LIN {X 0,Y 169.42,Z 430.477,A -85,B 0,C 180,E1 -24406.881,E2 -24406.881} C_VEL
LIN {X 0,Y 171.405,Z 398.166,A -85,B 0,C 180,E1 -24408.159,E2 -24408.159} C_VEL
LIN {X 0,Y 167.456,Z 387.202,A -85,B 0,C 180,E1 -24409.755,E2 -24409.755} C_VEL
LIN {X 0,Y 162.676,Z 376.705,A -85,B 0,C 180,E1 -24411.669,E2 -24411.669} C_VEL
LIN {X 0,Y 156.183,Z 365.5,A -85,B 0,C 180,E1 -24414.347,E2 -24414.347} C_VEL
LIN {X 0,Y 150.616,Z 356.98,A -85,B 0,C 180,E1 -24416.81,E2 -24416.81} C_VEL
LIN {X 0,Y 148.688,Z 354.013,A -85,B 0,C 180,E1 -24417.73,E2 -24417.73} C_VEL
LIN {X 0,Y 146.46,Z 350.663,A -85,B 0,C 180,E1 -24418.836,E2 -24418.836} C_VEL
LIN {X 0,Y 143.8,Z 347.278,A -85,B 0,C 180,E1 -24420.188,E2 -24420.188} C_VEL
LIN {X 0,Y 143.258,Z 345.674,A -85,B 0,C 180,E1 -24420.838,E2 -24420.838} C_VEL
LIN {X 0,Y 143.168,Z 345.197,A -85,B 0,C 180,E1 -24421.462,E2 -24421.462} C_VEL
LIN {X 0,Y 143.113,Z 345.14,A -85,B 0,C 180,E1 -24426.108,E2 -24426.108} C_VEL
LIN {X 0,Y 143.077,Z 345.141,A -85,B 0,C 180,E1 -24429.685,E2 -24429.685} C_VEL
LIN {X 0,Y 143.059,Z 345.139,A -85,B 0,C 180,E1 -24433.454,E2 -24433.454} C_VEL
LIN {X 0,Y 143.067,Z 345.145,A -85,B 0,C 180,E1 -24437.465,E2 -24437.465} C_VEL
LIN {X 0,Y 143.079,Z 345.123,A -85,B 0,C 180,E1 -24441.806,E2 -24441.806} C_VEL
LIN {X 0,Y 143.178,Z 345.126,A -85,B 0,C 180,E1 -24447.319,E2 -24447.319} C_VEL
LIN {X 0,Y 143.184,Z 345.102,A -85,B 0,C 180,E1 -24452.069,E2 -24452.069} C_VEL
LIN {X 0,Y 143.23,Z 345.111,A -85,B 0,C 180,E1 -24458.796,E2 -24458.796} C_VEL
LIN {X 0,Y 143.264,Z 345.082,A -85,B 0,C 180,E1 -24462.881,E2 -24462.881} C_VEL
LIN {X 0,Y 143.535,Z 345.1,A -85,B 0,C 180,E1 -24468.705,E2 -24468.705} C_VEL
LIN {X 0,Y 143.609,Z 345.048,A -85,B 0,C 180,E1 -24471.557,E2 -24471.557} C_VEL
LIN {X 0,Y 144.158,Z 345.024,A -85,B 0,C 180,E1 -24479.999,E2 -24479.999} C_VEL
LIN {X 0,Y 143.623,Z 345.077,A -85,B 0,C 180,E1 -24488.441,E2 -24488.441} C_VEL
LIN {X 0,Y 143.499,Z 345.099,A -85,B 0,C 180,E1 -24491.615,E2 -24491.615} C_VEL
LIN {X 0,Y 143.251,Z 345.109,A -85,B 0,C 180,E1 -24497.119,E2 -24497.119} C_VEL
LIN {X 0,Y 143.223,Z 345.13,A -85,B 0,C 180,E1 -24501.197,E2 -24501.197} C_VEL
LIN {X 0,Y 143.183,Z 345.151,A -85,B 0,C 180,E1 -24507.93,E2 -24507.93} C_VEL
LIN {X 0,Y 143.158,Z 345.189,A -85,B 0,C 180,E1 -24514.25,E2 -24514.25} C_VEL
LIN {X 0,Y 143.258,Z 345.961,A -85,B 0,C 180,E1 -24515.138,E2 -24515.138} C_VEL
LIN {X 0,Y 144.692,Z 348.88,A -85,B 0,C 180,E1 -24516.138,E2 -24516.138} C_VEL
LIN {X 0,Y 146.266,Z 350.451,A -85,B 0,C 180,E1 -24516.897,E2 -24516.897} C_VEL
LIN {X 0,Y 148.435,Z 353.858,A -85,B 0,C 180,E1 -24517.989,E2 -24517.989} C_VEL
LIN {X 0,Y 149.674,Z 355.677,A -85,B 0,C 180,E1 -24518.581,E2 -24518.581} C_VEL
LIN {X 0,Y 154.684,Z 363.406,A -85,B 0,C 180,E1 -24520.852,E2 -24520.852} C_VEL
LIN {X 0,Y 159.853,Z 373.317,A -85,B 0,C 180,E1 -24523.121,E2 -24523.121} C_VEL
LIN {X 0,Y 165.254,Z 385.644,A -85,B 0,C 180,E1 -24525.399,E2 -24525.399} C_VEL
LIN {X 0,Y 170.967,Z 401.167,A -85,B 0,C 180,E1 -24527.725,E2 -24527.725} C_VEL
LIN {X 0,Y 171.216,Z 402.78,A -85,B 0,C 180,E1 -24527.873,E2 -24527.873} C_VEL
LIN {X 0,Y 168.233,Z 448.35,A -85,B 0,C 180,E1 -24529.719,E2 -24529.719} C_VEL
LIN {X 0,Y 167.173,Z 458.294,A -85,B 0,C 180,E1 -24530.339,E2 -24530.339} C_VEL
LIN {X 0,Y 165.56,Z 468.543,A -85,B 0,C 180,E1 -24531.234,E2 -24531.234} C_VEL
LIN {X 0,Y 163.658,Z 477.716,A -85,B 0,C 180,E1 -24532.27,E2 -24532.27} C_VEL
LIN {X 0,Y 161.167,Z 488.501,A -85,B 0,C 180,E1 -24533.935,E2 -24533.935} C_VEL
LIN {X 0,Y 158.212,Z 498.547,A -85,B 0,C 180,E1 -24535.887,E2 -24535.887} C_VEL
LIN {X 0,Y 155.117,Z 507.96,A -85,B 0,C 180,E1 -24538.217,E2 -24538.217} C_VEL
LIN {X 0,Y 152.756,Z 515.01,A -85,B 0,C 180,E1 -24540.357,E2 -24540.357} C_VEL
LIN {X 0,Y 149.485,Z 523.905,A -85,B 0,C 180,E1 -24543.758,E2 -24543.758} C_VEL
LIN {X 0,Y 147.045,Z 530.294,A -85,B 0,C 180,E1 -24546.777,E2 -24546.777} C_VEL
LIN {X 0,Y 144.875,Z 536.086,A -85,B 0,C 180,E1 -24550.149,E2 -24550.149} C_VEL
LIN {X 0,Y 142.805,Z 541.677,A -85,B 0,C 180,E1 -24554.295,E2 -24554.295} C_VEL
LIN {X 0,Y 141.487,Z 546.063,A -85,B 0,C 180,E1 -24558.539,E2 -24558.539} C_VEL
LIN {X 0,Y 140.923,Z 548.391,A -85,B 0,C 180,E1 -24561.395,E2 -24561.395} C_VEL
LIN {X 0,Y 140.424,Z 551.696,A -85,B 0,C 180,E1 -24567.274,E2 -24567.274} C_VEL
LIN {X 0,Y 139.703,Z 552.498,A -85,B 0,C 180,E1 -24569.651,E2 -24569.651} C_VEL
LIN {X 0,Y 138.124,Z 553.012,A -85,B 0,C 180,E1 -24572.007,E2 -24572.007} C_VEL
LIN {X 0,Y 134.717,Z 553.305,A -85,B 0,C 180,E1 -24576.843,E2 -24576.843} C_VEL
LIN {X 0,Y 134.06,Z 553.015,A -85,B 0,C 180,E1 -24579.375,E2 -24579.375} C_VEL
LIN {X 0,Y 134.148,Z 552.859,A -85,B 0,C 180,E1 -24580.224,E2 -24580.224} C_VEL
LIN {X 0,Y 135.606,Z 551.577,A -85,B 0,C 180,E1 -24585.018,E2 -24585.018} C_VEL
LIN {X 0,Y 138.515,Z 548.533,A -85,B 0,C 180,E1 -24590.803,E2 -24590.803} C_VEL
LIN {X 0,Y 141.774,Z 545.076,A -85,B 0,C 180,E1 -24594.92,E2 -24594.92} C_VEL
LIN {X 0,Y 145.584,Z 540.569,A -85,B 0,C 180,E1 -24598.865,E2 -24598.865} C_VEL
LIN {X 0,Y 150.668,Z 533.867,A -85,B 0,C 180,E1 -24603.156,E2 -24603.156} C_VEL
LIN {X 0,Y 155.126,Z 527.779,A -85,B 0,C 180,E1 -24606.083,E2 -24606.083} C_VEL
LIN {X 0,Y 159.759,Z 520.62,A -85,B 0,C 180,E1 -24608.82,E2 -24608.82} C_VEL
LIN {X 0,Y 164.818,Z 511.938,A -85,B 0,C 180,E1 -24611.371,E2 -24611.371} C_VEL
LIN {X 0,Y 169.744,Z 502.444,A -85,B 0,C 180,E1 -24613.498,E2 -24613.498} C_VEL
LIN {X 0,Y 173.661,Z 493.629,A -85,B 0,C 180,E1 -24615.09,E2 -24615.09} C_VEL
LIN {X 0,Y 177.16,Z 484.552,A -85,B 0,C 180,E1 -24616.384,E2 -24616.384} C_VEL
LIN {X 0,Y 180.708,Z 473.055,A -85,B 0,C 180,E1 -24617.641,E2 -24617.641} C_VEL
LIN {X 0,Y 183.45,Z 461.877,A -85,B 0,C 180,E1 -24618.506,E2 -24618.506} C_VEL
LIN {X 0,Y 185.418,Z 450.53,A -85,B 0,C 180,E1 -24619.129,E2 -24619.129} C_VEL
LIN {X 0,Y 187.313,Z 431.246,A -85,B 0,C 180,E1 -24619.859,E2 -24619.859} C_VEL
LIN {X 0,Y 188.443,Z 418.099,A -85,B 0,C 180,E1 -24620.308,E2 -24620.308} C_VEL
LIN {X 0,Y 185.471,Z 410.111,A -85,B 0,C 180,E1 -24622.466,E2 -24622.466} C_VEL
LIN {X 0,Y 181.792,Z 401.756,A -85,B 0,C 180,E1 -24625.407,E2 -24625.407} C_VEL
LIN {X 0,Y 178.228,Z 394.65,A -85,B 0,C 180,E1 -24628.667,E2 -24628.667} C_VEL
LIN {X 0,Y 176.004,Z 390.795,A -85,B 0,C 180,E1 -24631.014,E2 -24631.014} C_VEL
LIN {X 0,Y 173.429,Z 386.846,A -85,B 0,C 180,E1 -24634.224,E2 -24634.224} C_VEL
LIN {X 0,Y 171.067,Z 383.644,A -85,B 0,C 180,E1 -24638.018,E2 -24638.018} C_VEL
LIN {X 0,Y 170.413,Z 382.188,A -85,B 0,C 180,E1 -24639.565,E2 -24639.565} C_VEL
LIN {X 0,Y 168.485,Z 380.243,A -85,B 0,C 180,E1 -24647.962,E2 -24647.962} C_VEL
LIN {X 0,Y 168.748,Z 380.458,A -85,B 0,C 180,E1 -24651.166,E2 -24651.166} C_VEL
LIN {X 0,Y 170.973,Z 382.26,A -85,B 0,C 180,E1 -24657.74,E2 -24657.74} C_VEL
LIN {X 0,Y 172.71,Z 385.701,A -85,B 0,C 180,E1 -24660.96,E2 -24660.96} C_VEL
LIN {X 0,Y 174.238,Z 387.45,A -85,B 0,C 180,E1 -24663.03,E2 -24663.03} C_VEL
LIN {X 0,Y 176.879,Z 391.787,A -85,B 0,C 180,E1 -24666.13,E2 -24666.13} C_VEL
LIN {X 0,Y 179.803,Z 396.635,A -85,B 0,C 180,E1 -24668.996,E2 -24668.996} C_VEL
LIN {X 0,Y 183.75,Z 403.362,A -85,B 0,C 180,E1 -24672.204,E2 -24672.204} C_VEL
LIN {X 0,Y 187.337,Z 411.633,A -85,B 0,C 180,E1 -24674.887,E2 -24674.887} C_VEL
LIN {X 0,Y 188.71,Z 415.167,A -85,B 0,C 180,E1 -24675.847,E2 -24675.847} C_VEL
LIN {X 0,Y 185.895,Z 445.064,A -85,B 0,C 180,E1 -24676.866,E2 -24676.866} C_VEL
LIN {X 0,Y 184.526,Z 454.52,A -85,B 0,C 180,E1 -24677.341,E2 -24677.341} C_VEL
LIN {X 0,Y 182.323,Z 464.877,A -85,B 0,C 180,E1 -24678.036,E2 -24678.036} C_VEL
LIN {X 0,Y 179.311,Z 476.023,A -85,B 0,C 180,E1 -24679.133,E2 -24679.133} C_VEL
LIN {X 0,Y 176.115,Z 485.452,A -85,B 0,C 180,E1 -24680.318,E2 -24680.318} C_VEL
LIN {X 0,Y 172.274,Z 494.993,A -85,B 0,C 180,E1 -24681.86,E2 -24681.86} C_VEL
LIN {X 0,Y 168.027,Z 504.044,A -85,B 0,C 180,E1 -24683.722,E2 -24683.722} C_VEL
LIN {X 0,Y 163.812,Z 511.888,A -85,B 0,C 180,E1 -24685.716,E2 -24685.716} C_VEL
LIN {X 0,Y 158.598,Z 520.414,A -85,B 0,C 180,E1 -24688.508,E2 -24688.508} C_VEL
LIN {X 0,Y 154.104,Z 526.971,A -85,B 0,C 180,E1 -24691.229,E2 -24691.229} C_VEL
LIN {X 0,Y 149.899,Z 532.66,A -85,B 0,C 180,E1 -24694.238,E2 -24694.238} C_VEL
LIN {X 0,Y 146.063,Z 537.442,A -85,B 0,C 180,E1 -24697.447,E2 -24697.447} C_VEL
LIN {X 0,Y 141.742,Z 542.341,A -85,B 0,C 180,E1 -24701.949,E2 -24701.949} C_VEL
LIN {X 0,Y 139.33,Z 544.911,A -85,B 0,C 180,E1 -24705.075,E2 -24705.075} C_VEL
LIN {X 0,Y 136.054,Z 547.988,A -85,B 0,C 180,E1 -24710.792,E2 -24710.792} C_VEL
LIN {X 0,Y 134.497,Z 549.246,A -85,B 0,C 180,E1 -24714.915,E2 -24714.915} C_VEL
LIN {X 0,Y 133.629,Z 549.592,A -85,B 0,C 180,E1 -24718.269,E2 -24718.269} C_VEL
LIN {X 0,Y 132.836,Z 549.037,A -85,B 0,C 180,E1 -24724.96,E2 -24724.96} C_VEL
LIN {X 0,Y 132.855,Z 547.969,A -85,B 0,C 180,E1 -24728.266,E2 -24728.266} C_VEL
LIN {X 0,Y 133.226,Z 546.339,A -85,B 0,C 180,E1 -24731.723,E2 -24731.723} C_VEL
LIN {X 0,Y 134.201,Z 543.282,A -85,B 0,C 180,E1 -24736.37,E2 -24736.37} C_VEL
LIN {X 0,Y 135.436,Z 539.701,A -85,B 0,C 180,E1 -24740.384,E2 -24740.384} C_VEL
LIN {X 0,Y 137.031,Z 535.472,A -85,B 0,C 180,E1 -24744.113,E2 -24744.113} C_VEL
LIN {X 0,Y 139.182,Z 530.061,A -85,B 0,C 180,E1 -24747.902,E2 -24747.902} C_VEL
LIN {X 0,Y 141.754,Z 523.767,A -85,B 0,C 180,E1 -24751.421,E2 -24751.421} C_VEL
LIN {X 0,Y 144.817,Z 515.992,A -85,B 0,C 180,E1 -24754.872,E2 -24754.872} C_VEL
LIN {X 0,Y 147.942,Z 507.566,A -85,B 0,C 180,E1 -24757.85,E2 -24757.85} C_VEL
LIN {X 0,Y 150.993,Z 499.018,A -85,B 0,C 180,E1 -24760.252,E2 -24760.252} C_VEL
LIN {X 0,Y 153.669,Z 490.48,A -85,B 0,C 180,E1 -24762.212,E2 -24762.212} C_VEL
LIN {X 0,Y 156.274,Z 480.837,A -85,B 0,C 180,E1 -24763.989,E2 -24763.989} C_VEL
LIN {X 0,Y 158.85,Z 469.502,A -85,B 0,C 180,E1 -24765.575,E2 -24765.575} C_VEL
LIN {X 0,Y 160.694,Z 458.708,A -85,B 0,C 180,E1 -24766.72,E2 -24766.72} C_VEL
LIN {X 0,Y 162.232,Z 447.473,A -85,B 0,C 180,E1 -24767.521,E2 -24767.521} C_VEL
LIN {X 0,Y 163.725,Z 428.996,A -85,B 0,C 180,E1 -24768.341,E2 -24768.341} C_VEL
LIN {X 0,Y 165.514,Z 399.768,A -85,B 0,C 180,E1 -24769.546,E2 -24769.546} C_VEL
LIN {X 0,Y 161.92,Z 389.844,A -85,B 0,C 180,E1 -24771.101,E2 -24771.101} C_VEL
LIN {X 0,Y 157.712,Z 380.464,A -85,B 0,C 180,E1 -24772.916,E2 -24772.916} C_VEL
LIN {X 0,Y 151.583,Z 369.812,A -85,B 0,C 180,E1 -24775.593,E2 -24775.593} C_VEL
LIN {X 0,Y 145.009,Z 359.507,A -85,B 0,C 180,E1 -24778.765,E2 -24778.765} C_VEL
LIN {X 0,Y 141.709,Z 354.853,A -85,B 0,C 180,E1 -24780.492,E2 -24780.492} C_VEL
LIN {X 0,Y 139.638,Z 351.74,A -85,B 0,C 180,E1 -24781.645,E2 -24781.645} C_VEL
LIN {X 0,Y 138.864,Z 350.808,A -85,B 0,C 180,E1 -24782.071,E2 -24782.071} C_VEL
LIN {X 0,Y 136.849,Z 348.327,A -85,B 0,C 180,E1 -24783.225,E2 -24783.225} C_VEL
LIN {X 0,Y 136.198,Z 346.577,A -85,B 0,C 180,E1 -24783.99,E2 -24783.99} C_VEL
LIN {X 0,Y 136.082,Z 346.085,A -85,B 0,C 180,E1 -24784.618,E2 -24784.618} C_VEL
LIN {X 0,Y 136.053,Z 346.02,A -85,B 0,C 180,E1 -24789.208,E2 -24789.208} C_VEL
LIN {X 0,Y 136.001,Z 346.019,A -85,B 0,C 180,E1 -24793.658,E2 -24793.658} C_VEL
LIN {X 0,Y 136.007,Z 346.018,A -85,B 0,C 180,E1 -24797.796,E2 -24797.796} C_VEL
LIN {X 0,Y 136.028,Z 346,A -85,B 0,C 180,E1 -24801.684,E2 -24801.684} C_VEL
LIN {X 0,Y 136.085,Z 346.032,A -85,B 0,C 180,E1 -24805.722,E2 -24805.722} C_VEL
LIN {X 0,Y 136.125,Z 345.982,A -85,B 0,C 180,E1 -24812.311,E2 -24812.311} C_VEL
LIN {X 0,Y 136.196,Z 345.984,A -85,B 0,C 180,E1 -24818.824,E2 -24818.824} C_VEL
LIN {X 0,Y 136.234,Z 345.98,A -85,B 0,C 180,E1 -24825.051,E2 -24825.051} C_VEL
LIN {X 0,Y 136.427,Z 345.989,A -85,B 0,C 180,E1 -24828.177,E2 -24828.177} C_VEL
LIN {X 0,Y 136.538,Z 345.933,A -85,B 0,C 180,E1 -24831.116,E2 -24831.116} C_VEL
LIN {X 0,Y 137.115,Z 345.901,A -85,B 0,C 180,E1 -24839.999,E2 -24839.999} C_VEL
LIN {X 0,Y 136.549,Z 345.964,A -85,B 0,C 180,E1 -24848.882,E2 -24848.882} C_VEL
LIN {X 0,Y 136.414,Z 345.975,A -85,B 0,C 180,E1 -24851.892,E2 -24851.892} C_VEL
LIN {X 0,Y 136.165,Z 346.002,A -85,B 0,C 180,E1 -24858.039,E2 -24858.039} C_VEL
LIN {X 0,Y 136.148,Z 346.003,A -85,B 0,C 180,E1 -24861.694,E2 -24861.694} C_VEL
LIN {X 0,Y 136.092,Z 346.024,A -85,B 0,C 180,E1 -24868.608,E2 -24868.608} C_VEL
LIN {X 0,Y 136.09,Z 346.281,A -85,B 0,C 180,E1 -24871.525,E2 -24871.525} C_VEL
LIN {X 0,Y 136.445,Z 347.466,A -85,B 0,C 180,E1 -24872.302,E2 -24872.302} C_VEL
LIN {X 0,Y 138.171,Z 350.216,A -85,B 0,C 180,E1 -24873.384,E2 -24873.384} C_VEL
LIN {X 0,Y 139.409,Z 351.47,A -85,B 0,C 180,E1 -24874.054,E2 -24874.054} C_VEL
LIN {X 0,Y 141.532,Z 354.861,A -85,B 0,C 180,E1 -24875.257,E2 -24875.257} C_VEL
LIN {X 0,Y 143.129,Z 357.003,A -85,B 0,C 180,E1 -24876.101,E2 -24876.101} C_VEL
LIN {X 0,Y 148.206,Z 364.638,A -85,B 0,C 180,E1 -24878.667,E2 -24878.667} C_VEL
LIN {X 0,Y 152.246,Z 371.513,A -85,B 0,C 180,E1 -24880.573,E2 -24880.573} C_VEL
LIN {X 0,Y 157.962,Z 383.796,A -85,B 0,C 180,E1 -24883.197,E2 -24883.197} C_VEL
LIN {X 0,Y 163.187,Z 397.335,A -85,B 0,C 180,E1 -24885.518,E2 -24885.518} C_VEL
LIN {X 0,Y 165.396,Z 403.646,A -85,B 0,C 180,E1 -24886.469,E2 -24886.469} C_VEL
LIN {X 0,Y 162.325,Z 448.845,A -85,B 0,C 180,E1 -24888.358,E2 -24888.358} C_VEL
LIN {X 0,Y 161.232,Z 458.516,A -85,B 0,C 180,E1 -24888.987,E2 -24888.987} C_VEL
LIN {X 0,Y 159.578,Z 468.651,A -85,B 0,C 180,E1 -24889.901,E2 -24889.901} C_VEL
LIN {X 0,Y 157.602,Z 477.772,A -85,B 0,C 180,E1 -24890.958,E2 -24890.958} C_VEL
LIN {X 0,Y 155.005,Z 488.528,A -85,B 0,C 180,E1 -24892.668,E2 -24892.668} C_VEL
LIN {X 0,Y 151.935,Z 498.551,A -85,B 0,C 180,E1 -24894.675,E2 -24894.675} C_VEL
LIN {X 0,Y 148.705,Z 507.945,A -85,B 0,C 180,E1 -24897.077,E2 -24897.077} C_VEL
LIN {X 0,Y 145.899,Z 515.846,A -85,B 0,C 180,E1 -24899.616,E2 -24899.616} C_VEL
LIN {X 0,Y 142.775,Z 523.96,A -85,B 0,C 180,E1 -24902.871,E2 -24902.871} C_VEL
LIN {X 0,Y 139.995,Z 530.839,A -85,B 0,C 180,E1 -24906.321,E2 -24906.321} C_VEL
LIN {X 0,Y 138.164,Z 535.532,A -85,B 0,C 180,E1 -24909.141,E2 -24909.141} C_VEL
LIN {X 0,Y 135.935,Z 541.224,A -85,B 0,C 180,E1 -24913.479,E2 -24913.479} C_VEL
LIN {X 0,Y 134.51,Z 545.696,A -85,B 0,C 180,E1 -24917.936,E2 -24917.936} C_VEL
LIN {X 0,Y 133.889,Z 548.023,A -85,B 0,C 180,E1 -24920.939,E2 -24920.939} C_VEL
LIN {X 0,Y 133.332,Z 551.432,A -85,B 0,C 180,E1 -24926.978,E2 -24926.978} C_VEL
LIN {X 0,Y 133.415,Z 552.393,A -85,B 0,C 180,E1 -24930,E2 -24930} C_VEL
LIN {X 0,Y 133.515,Z 553.311,A -85,B 0,C 180,E1 -24936.043,E2 -24936.043} C_VEL
LIN {X 0,Y 134.148,Z 552.859,A -85,B 0,C 180,E1 -24940.224,E2 -24940.224} C_VEL
LIN {X 0,Y 134.121,Z 552.393,A -85,B 0,C 180,E1 -24942.742,E2 -24942.742} C_VEL
LIN {X 0,Y 132.78,Z 551.096,A -85,B 0,C 180,E1 -24946.934,E2 -24946.934} C_VEL
LIN {X 0,Y 132.116,Z 549.103,A -85,B 0,C 180,E1 -24951.129,E2 -24951.129} C_VEL
LIN {X 0,Y 133.122,Z 547.442,A -85,B 0,C 180,E1 -24953.54,E2 -24953.54} C_VEL
LIN {X 0,Y 136.723,Z 543.887,A -85,B 0,C 180,E1 -24957.557,E2 -24957.557} C_VEL
LIN {X 0,Y 140.881,Z 539.102,A -85,B 0,C 180,E1 -24961.587,E2 -24961.587} C_VEL
LIN {X 0,Y 145.729,Z 533.082,A -85,B 0,C 180,E1 -24965.36,E2 -24965.36} C_VEL
LIN {X 0,Y 150.396,Z 527.009,A -85,B 0,C 180,E1 -24968.255,E2 -24968.255} C_VEL
LIN {X 0,Y 155.42,Z 519.728,A -85,B 0,C 180,E1 -24970.971,E2 -24970.971} C_VEL
LIN {X 0,Y 160.705,Z 510.929,A -85,B 0,C 180,E1 -24973.534,E2 -24973.534} C_VEL
LIN {X 0,Y 165.299,Z 502.475,A -85,B 0,C 180,E1 -24975.41,E2 -24975.41} C_VEL
LIN {X 0,Y 169.386,Z 493.684,A -85,B 0,C 180,E1 -24976.994,E2 -24976.994} C_VEL
LIN {X 0,Y 173.603,Z 482.834,A -85,B 0,C 180,E1 -24978.498,E2 -24978.498} C_VEL
LIN {X 0,Y 176.583,Z 473.688,A -85,B 0,C 180,E1 -24979.474,E2 -24979.474} C_VEL
LIN {X 0,Y 179.612,Z 461.78,A -85,B 0,C 180,E1 -24980.392,E2 -24980.392} C_VEL
LIN {X 0,Y 181.585,Z 450.908,A -85,B 0,C 180,E1 -24980.988,E2 -24980.988} C_VEL
LIN {X 0,Y 183.476,Z 432.692,A -85,B 0,C 180,E1 -24981.682,E2 -24981.682} C_VEL
LIN {X 0,Y 184.515,Z 420.712,A -85,B 0,C 180,E1 -24982.108,E2 -24982.108} C_VEL
LIN {X 0,Y 181.36,Z 412.254,A -85,B 0,C 180,E1 -24984.694,E2 -24984.694} C_VEL
LIN {X 0,Y 178.028,Z 404.613,A -85,B 0,C 180,E1 -24987.713,E2 -24987.713} C_VEL
LIN {X 0,Y 175.056,Z 398.582,A -85,B 0,C 180,E1 -24990.874,E2 -24990.874} C_VEL
LIN {X 0,Y 173.509,Z 396.227,A -85,B 0,C 180,E1 -24992.688,E2 -24992.688} C_VEL
LIN {X 0,Y 171.894,Z 393.442,A -85,B 0,C 180,E1 -24994.974,E2 -24994.974} C_VEL
LIN {X 0,Y 169.789,Z 390.364,A -85,B 0,C 180,E1 -24998.654,E2 -24998.654} C_VEL
LIN {X 0,Y 169.326,Z 389.162,A -85,B 0,C 180,E1 -24999.853,E2 -24999.853} C_VEL
LIN {X 0,Y 167.545,Z 387.302,A -85,B 0,C 180,E1 -25007.894,E2 -25007.894} C_VEL
LIN {X 0,Y 167.798,Z 387.503,A -85,B 0,C 180,E1 -25011.116,E2 -25011.116} C_VEL
LIN {X 0,Y 169.735,Z 389.122,A -85,B 0,C 180,E1 -25017.182,E2 -25017.182} C_VEL
LIN {X 0,Y 171.478,Z 392.631,A -85,B 0,C 180,E1 -25020.605,E2 -25020.605} C_VEL
LIN {X 0,Y 172.688,Z 394.127,A -85,B 0,C 180,E1 -25022.333,E2 -25022.333} C_VEL
LIN {X 0,Y 175.084,Z 398.253,A -85,B 0,C 180,E1 -25025.358,E2 -25025.358} C_VEL
LIN {X 0,Y 177.855,Z 403.08,A -85,B 0,C 180,E1 -25028.234,E2 -25028.234} C_VEL
LIN {X 0,Y 181.051,Z 408.824,A -85,B 0,C 180,E1 -25031.037,E2 -25031.037} C_VEL
LIN {X 0,Y 184.2,Z 416.496,A -85,B 0,C 180,E1 -25033.615,E2 -25033.615} C_VEL
LIN {X 0,Y 184.757,Z 418.082,A -85,B 0,C 180,E1 -25034.057,E2 -25034.057} C_VEL
LIN {X 0,Y 182.12,Z 445.2,A -85,B 0,C 180,E1 -25034.994,E2 -25034.994} C_VEL
LIN {X 0,Y 180.59,Z 455.19,A -85,B 0,C 180,E1 -25035.496,E2 -25035.496} C_VEL
LIN {X 0,Y 178.403,Z 465.096,A -85,B 0,C 180,E1 -25036.162,E2 -25036.162} C_VEL
LIN {X 0,Y 175.245,Z 476.308,A -85,B 0,C 180,E1 -25037.26,E2 -25037.26} C_VEL
LIN {X 0,Y 172.143,Z 485.121,A -85,B 0,C 180,E1 -25038.338,E2 -25038.338} C_VEL
LIN {X 0,Y 167.782,Z 495.487,A -85,B 0,C 180,E1 -25040.013,E2 -25040.013} C_VEL
LIN {X 0,Y 163.619,Z 503.956,A -85,B 0,C 180,E1 -25041.741,E2 -25041.741} C_VEL
LIN {X 0,Y 159.181,Z 511.899,A -85,B 0,C 180,E1 -25043.774,E2 -25043.774} C_VEL
LIN {X 0,Y 153.572,Z 520.561,A -85,B 0,C 180,E1 -25046.628,E2 -25046.628} C_VEL
LIN {X 0,Y 149.027,Z 526.848,A -85,B 0,C 180,E1 -25049.256,E2 -25049.256} C_VEL
LIN {X 0,Y 144.444,Z 532.653,A -85,B 0,C 180,E1 -25052.359,E2 -25052.359} C_VEL
LIN {X 0,Y 139.573,Z 538.241,A -85,B 0,C 180,E1 -25056.327,E2 -25056.327} C_VEL
LIN {X 0,Y 136.454,Z 541.627,A -85,B 0,C 180,E1 -25059.415,E2 -25059.415} C_VEL
LIN {X 0,Y 133.247,Z 544.766,A -85,B 0,C 180,E1 -25063.29,E2 -25063.29} C_VEL
LIN {X 0,Y 129.46,Z 548.058,A -85,B 0,C 180,E1 -25069.467,E2 -25069.467} C_VEL
LIN {X 0,Y 128.013,Z 549.08,A -85,B 0,C 180,E1 -25072.85,E2 -25072.85} C_VEL
LIN {X 0,Y 126.957,Z 549.594,A -85,B 0,C 180,E1 -25076.388,E2 -25076.388} C_VEL
LIN {X 0,Y 126.176,Z 549.719,A -85,B 0,C 180,E1 -25079.914,E2 -25079.914} C_VEL
LIN {X 0,Y 125.801,Z 549.344,A -85,B 0,C 180,E1 -25083.454,E2 -25083.454} C_VEL
LIN {X 0,Y 125.943,Z 547.072,A -85,B 0,C 180,E1 -25090.439,E2 -25090.439} C_VEL
LIN {X 0,Y 126.87,Z 544.129,A -85,B 0,C 180,E1 -25095.566,E2 -25095.566} C_VEL
LIN {X 0,Y 127.789,Z 541.636,A -85,B 0,C 180,E1 -25098.904,E2 -25098.904} C_VEL
LIN {X 0,Y 129.998,Z 535.778,A -85,B 0,C 180,E1 -25104.571,E2 -25104.571} C_VEL
LIN {X 0,Y 132.201,Z 530.534,A -85,B 0,C 180,E1 -25108.477,E2 -25108.477} C_VEL
LIN {X 0,Y 134.983,Z 524.035,A -85,B 0,C 180,E1 -25112.305,E2 -25112.305} C_VEL
LIN {X 0,Y 138.151,Z 516.445,A -85,B 0,C 180,E1 -25115.84,E2 -25115.84} C_VEL
LIN {X 0,Y 141.565,Z 507.662,A -85,B 0,C 180,E1 -25119.069,E2 -25119.069} C_VEL
LIN {X 0,Y 144.745,Z 499.104,A -85,B 0,C 180,E1 -25121.554,E2 -25121.554} C_VEL
LIN {X 0,Y 147.786,Z 489.659,A -85,B 0,C 180,E1 -25123.756,E2 -25123.756} C_VEL
LIN {X 0,Y 150.559,Z 479.769,A -85,B 0,C 180,E1 -25125.57,E2 -25125.57} C_VEL
LIN {X 0,Y 152.965,Z 469.48,A -85,B 0,C 180,E1 -25127.032,E2 -25127.032} C_VEL
LIN {X 0,Y 154.859,Z 458.89,A -85,B 0,C 180,E1 -25128.181,E2 -25128.181} C_VEL
LIN {X 0,Y 156.412,Z 448.069,A -85,B 0,C 180,E1 -25128.978,E2 -25128.978} C_VEL
LIN {X 0,Y 157.946,Z 430.09,A -85,B 0,C 180,E1 -25129.8,E2 -25129.8} C_VEL
LIN {X 0,Y 159.769,Z 401.488,A -85,B 0,C 180,E1 -25131.012,E2 -25131.012} C_VEL
LIN {X 0,Y 155.979,Z 391.113,A -85,B 0,C 180,E1 -25132.78,E2 -25132.78} C_VEL
LIN {X 0,Y 152.062,Z 382.89,A -85,B 0,C 180,E1 -25134.555,E2 -25134.555} C_VEL
LIN {X 0,Y 146.807,Z 373.79,A -85,B 0,C 180,E1 -25137.033,E2 -25137.033} C_VEL
LIN {X 0,Y 141.181,Z 364.71,A -85,B 0,C 180,E1 -25139.948,E2 -25139.948} C_VEL
LIN {X 0,Y 137.751,Z 359.893,A -85,B 0,C 180,E1 -25141.842,E2 -25141.842} C_VEL
LIN {X 0,Y 135.354,Z 356.36,A -85,B 0,C 180,E1 -25143.273,E2 -25143.273} C_VEL
LIN {X 0,Y 133.051,Z 353.187,A -85,B 0,C 180,E1 -25144.718,E2 -25144.718} C_VEL
LIN {X 0,Y 132.328,Z 352.128,A -85,B 0,C 180,E1 -25145.197,E2 -25145.197} C_VEL
LIN {X 0,Y 130.053,Z 349.935,A -85,B 0,C 180,E1 -25146.666,E2 -25146.666} C_VEL
LIN {X 0,Y 129.128,Z 347.688,A -85,B 0,C 180,E1 -25147.641,E2 -25147.641} C_VEL
LIN {X 0,Y 129.016,Z 346.961,A -85,B 0,C 180,E1 -25148.541,E2 -25148.541} C_VEL
LIN {X 0,Y 128.924,Z 346.919,A -85,B 0,C 180,E1 -25155.127,E2 -25155.127} C_VEL
LIN {X 0,Y 128.944,Z 346.879,A -85,B 0,C 180,E1 -25159.735,E2 -25159.735} C_VEL
LIN {X 0,Y 128.982,Z 346.916,A -85,B 0,C 180,E1 -25164.818,E2 -25164.818} C_VEL
LIN {X 0,Y 129.018,Z 346.859,A -85,B 0,C 180,E1 -25170.642,E2 -25170.642} C_VEL
LIN {X 0,Y 129.016,Z 346.89,A -85,B 0,C 180,E1 -25174.164,E2 -25174.164} C_VEL
LIN {X 0,Y 129.075,Z 346.888,A -85,B 0,C 180,E1 -25177.765,E2 -25177.765} C_VEL
LIN {X 0,Y 129.154,Z 346.849,A -85,B 0,C 180,E1 -25184.211,E2 -25184.211} C_VEL
LIN {X 0,Y 129.347,Z 346.871,A -85,B 0,C 180,E1 -25187.967,E2 -25187.967} C_VEL
LIN {X 0,Y 129.464,Z 346.819,A -85,B 0,C 180,E1 -25190.627,E2 -25190.627} C_VEL
LIN {X 0,Y 130.07,Z 346.778,A -85,B 0,C 180,E1 -25199.999,E2 -25199.999} C_VEL
LIN {X 0,Y 129.471,Z 346.852,A -85,B 0,C 180,E1 -25209.371,E2 -25209.371} C_VEL
LIN {X 0,Y 129.298,Z 346.85,A -85,B 0,C 180,E1 -25212.557,E2 -25212.557} C_VEL
LIN {X 0,Y 129.084,Z 346.9,A -85,B 0,C 180,E1 -25219.066,E2 -25219.066} C_VEL
LIN {X 0,Y 129.045,Z 346.88,A -85,B 0,C 180,E1 -25222.409,E2 -25222.409} C_VEL
LIN {X 0,Y 129.095,Z 347.029,A -85,B 0,C 180,E1 -25227.563,E2 -25227.563} C_VEL
LIN {X 0,Y 129.358,Z 348.214,A -85,B 0,C 180,E1 -25228.533,E2 -25228.533} C_VEL
LIN {X 0,Y 130.768,Z 350.777,A -85,B 0,C 180,E1 -25229.647,E2 -25229.647} C_VEL
LIN {X 0,Y 132.707,Z 352.512,A -85,B 0,C 180,E1 -25230.866,E2 -25230.866} C_VEL
LIN {X 0,Y 134.929,Z 355.991,A -85,B 0,C 180,E1 -25232.311,E2 -25232.311} C_VEL
LIN {X 0,Y 136.097,Z 357.553,A -85,B 0,C 180,E1 -25233.013,E2 -25233.013} C_VEL
LIN {X 0,Y 141.892,Z 366.04,A -85,B 0,C 180,E1 -25236.274,E2 -25236.274} C_VEL
LIN {X 0,Y 147.239,Z 374.845,A -85,B 0,C 180,E1 -25239.029,E2 -25239.029} C_VEL
LIN {X 0,Y 153.048,Z 387.457,A -85,B 0,C 180,E1 -25241.892,E2 -25241.892} C_VEL
LIN {X 0,Y 158.407,Z 401.74,A -85,B 0,C 180,E1 -25244.437,E2 -25244.437} C_VEL
LIN {X 0,Y 159.627,Z 405.36,A -85,B 0,C 180,E1 -25245.007,E2 -25245.007} C_VEL
LIN {X 0,Y 158.009,Z 430.26,A -85,B 0,C 180,E1 -25246.053,E2 -25246.053} C_VEL
LIN {X 0,Y 156.427,Z 450.314,A -85,B 0,C 180,E1 -25246.959,E2 -25246.959} C_VEL
LIN {X 0,Y 155.189,Z 460.064,A -85,B 0,C 180,E1 -25247.651,E2 -25247.651} C_VEL
LIN {X 0,Y 153.42,Z 469.897,A -85,B 0,C 180,E1 -25248.595,E2 -25248.595} C_VEL
LIN {X 0,Y 151.111,Z 479.645,A -85,B 0,C 180,E1 -25249.81,E2 -25249.81} C_VEL
LIN {X 0,Y 148.921,Z 488.522,A -85,B 0,C 180,E1 -25251.295,E2 -25251.295} C_VEL
LIN {X 0,Y 146.16,Z 497.288,A -85,B 0,C 180,E1 -25253.054,E2 -25253.054} C_VEL
LIN {X 0,Y 142.801,Z 506.887,A -85,B 0,C 180,E1 -25255.529,E2 -25255.529} C_VEL
LIN {X 0,Y 139.77,Z 514.938,A -85,B 0,C 180,E1 -25258.131,E2 -25258.131} C_VEL
LIN {X 0,Y 136.237,Z 523.593,A -85,B 0,C 180,E1 -25261.692,E2 -25261.692} C_VEL
LIN {X 0,Y 133.479,Z 530.184,A -85,B 0,C 180,E1 -25265.088,E2 -25265.088} C_VEL
LIN {X 0,Y 131.517,Z 534.929,A -85,B 0,C 180,E1 -25268.033,E2 -25268.033} C_VEL
LIN {X 0,Y 129.105,Z 540.75,A -85,B 0,C 180,E1 -25272.578,E2 -25272.578} C_VEL
LIN {X 0,Y 127.558,Z 545.318,A -85,B 0,C 180,E1 -25277.268,E2 -25277.268} C_VEL
LIN {X 0,Y 126.877,Z 547.653,A -85,B 0,C 180,E1 -25280.434,E2 -25280.434} C_VEL
LIN {X 0,Y 126.246,Z 551.192,A -85,B 0,C 180,E1 -25286.808,E2 -25286.808} C_VEL
LIN {X 0,Y 126.317,Z 552.181,A -85,B 0,C 180,E1 -25290,E2 -25290} C_VEL
LIN {X 0,Y 126.301,Z 552.877,A -85,B 0,C 180,E1 -25293.19,E2 -25293.19} C_VEL
LIN {X 0,Y 126.45,Z 553.175,A -85,B 0,C 180,E1 -25296.382,E2 -25296.382} C_VEL
LIN {X 0,Y 127.659,Z 552.569,A -85,B 0,C 180,E1 -25302.721,E2 -25302.721} C_VEL
LIN {X 0,Y 130.135,Z 550.298,A -85,B 0,C 180,E1 -25308.907,E2 -25308.907} C_VEL
LIN {X 0,Y 132.977,Z 547.592,A -85,B 0,C 180,E1 -25313.352,E2 -25313.352} C_VEL
LIN {X 0,Y 133.122,Z 547.442,A -85,B 0,C 180,E1 -25313.54,E2 -25313.54} C_VEL
LIN {X 0,Y 134.341,Z 545.697,A -85,B 0,C 180,E1 -25315.886,E2 -25315.886} C_VEL
LIN {X 0,Y 135.038,Z 542.326,A -85,B 0,C 180,E1 -25319.858,E2 -25319.858} C_VEL
LIN {X 0,Y 135.842,Z 539.39,A -85,B 0,C 180,E1 -25322.957,E2 -25322.957} C_VEL
LIN {X 0,Y 137.381,Z 536.737,A -85,B 0,C 180,E1 -25325.094,E2 -25325.094} C_VEL
LIN {X 0,Y 138.168,Z 535.792,A -85,B 0,C 180,E1 -25325.742,E2 -25325.742} C_VEL
LIN {X 0,Y 144.924,Z 527.69,A -85,B 0,C 180,E1 -25329.982,E2 -25329.982} C_VEL
LIN {X 0,Y 150.177,Z 520.561,A -85,B 0,C 180,E1 -25332.732,E2 -25332.732} C_VEL
LIN {X 0,Y 155.68,Z 511.945,A -85,B 0,C 180,E1 -25335.317,E2 -25335.317} C_VEL
LIN {X 0,Y 161.051,Z 502.506,A -85,B 0,C 180,E1 -25337.425,E2 -25337.425} C_VEL
LIN {X 0,Y 165.308,Z 493.74,A -85,B 0,C 180,E1 -25338.993,E2 -25338.993} C_VEL
LIN {X 0,Y 169.688,Z 482.96,A -85,B 0,C 180,E1 -25340.479,E2 -25340.479} C_VEL
LIN {X 0,Y 173.029,Z 473.013,A -85,B 0,C 180,E1 -25341.514,E2 -25341.514} C_VEL
LIN {X 0,Y 176.051,Z 461.469,A -85,B 0,C 180,E1 -25342.38,E2 -25342.38} C_VEL
LIN {X 0,Y 178.062,Z 450.767,A -85,B 0,C 180,E1 -25342.955,E2 -25342.955} C_VEL
LIN {X 0,Y 180.02,Z 432.886,A -85,B 0,C 180,E1 -25343.626,E2 -25343.626} C_VEL
LIN {X 0,Y 180.813,Z 423.539,A -85,B 0,C 180,E1 -25343.994,E2 -25343.994} C_VEL
LIN {X 0,Y 178.175,Z 416.369,A -85,B 0,C 180,E1 -25346.38,E2 -25346.38} C_VEL
LIN {X 0,Y 175.543,Z 409.985,A -85,B 0,C 180,E1 -25349.06,E2 -25349.06} C_VEL
LIN {X 0,Y 173.161,Z 404.746,A -85,B 0,C 180,E1 -25351.833,E2 -25351.833} C_VEL
LIN {X 0,Y 170.439,Z 400.163,A -85,B 0,C 180,E1 -25355.648,E2 -25355.648} C_VEL
LIN {X 0,Y 168.378,Z 396.657,A -85,B 0,C 180,E1 -25359.721,E2 -25359.721} C_VEL
LIN {X 0,Y 168.109,Z 396.046,A -85,B 0,C 180,E1 -25360.462,E2 -25360.462} C_VEL
LIN {X 0,Y 166.609,Z 394.333,A -85,B 0,C 180,E1 -25367.825,E2 -25367.825} C_VEL
LIN {X 0,Y 166.85,Z 394.532,A -85,B 0,C 180,E1 -25371.065,E2 -25371.065} C_VEL
LIN {X 0,Y 168.548,Z 396.094,A -85,B 0,C 180,E1 -25376.714,E2 -25376.714} C_VEL
LIN {X 0,Y 170.322,Z 399.643,A -85,B 0,C 180,E1 -25380.352,E2 -25380.352} C_VEL
LIN {X 0,Y 171.28,Z 400.987,A -85,B 0,C 180,E1 -25381.796,E2 -25381.796} C_VEL
LIN {X 0,Y 173.454,Z 404.973,A -85,B 0,C 180,E1 -25384.731,E2 -25384.731} C_VEL
LIN {X 0,Y 176.085,Z 409.753,A -85,B 0,C 180,E1 -25387.599,E2 -25387.599} C_VEL
LIN {X 0,Y 178.682,Z 414.897,A -85,B 0,C 180,E1 -25390.07,E2 -25390.07} C_VEL
LIN {X 0,Y 181.098,Z 421.021,A -85,B 0,C 180,E1 -25392.199,E2 -25392.199} C_VEL
LIN {X 0,Y 178.518,Z 446.025,A -85,B 0,C 180,E1 -25393.066,E2 -25393.066} C_VEL
LIN {X 0,Y 177.024,Z 455.271,A -85,B 0,C 180,E1 -25393.528,E2 -25393.528} C_VEL
LIN {X 0,Y 175.003,Z 464.336,A -85,B 0,C 180,E1 -25394.117,E2 -25394.117} C_VEL
LIN {X 0,Y 171.612,Z 475.961,A -85,B 0,C 180,E1 -25395.214,E2 -25395.214} C_VEL
LIN {X 0,Y 168.398,Z 484.846,A -85,B 0,C 180,E1 -25396.283,E2 -25396.283} C_VEL
LIN {X 0,Y 163.708,Z 495.516,A -85,B 0,C 180,E1 -25397.98,E2 -25397.98} C_VEL
LIN {X 0,Y 158.836,Z 504.894,A -85,B 0,C 180,E1 -25399.907,E2 -25399.907} C_VEL
LIN {X 0,Y 154.585,Z 512.129,A -85,B 0,C 180,E1 -25401.77,E2 -25401.77} C_VEL
LIN {X 0,Y 148.791,Z 520.665,A -85,B 0,C 180,E1 -25404.598,E2 -25404.598} C_VEL
LIN {X 0,Y 144.148,Z 526.773,A -85,B 0,C 180,E1 -25407.154,E2 -25407.154} C_VEL
LIN {X 0,Y 138.816,Z 533.08,A -85,B 0,C 180,E1 -25410.608,E2 -25410.608} C_VEL
LIN {X 0,Y 133.569,Z 538.658,A -85,B 0,C 180,E1 -25414.741,E2 -25414.741} C_VEL
LIN {X 0,Y 129.882,Z 542.313,A -85,B 0,C 180,E1 -25418.316,E2 -25418.316} C_VEL
LIN {X 0,Y 125.738,Z 545.941,A -85,B 0,C 180,E1 -25423.397,E2 -25423.397} C_VEL
LIN {X 0,Y 122.926,Z 548.133,A -85,B 0,C 180,E1 -25428.009,E2 -25428.009} C_VEL
LIN {X 0,Y 120.191,Z 549.658,A -85,B 0,C 180,E1 -25434.949,E2 -25434.949} C_VEL
LIN {X 0,Y 119.404,Z 549.905,A -85,B 0,C 180,E1 -25438.013,E2 -25438.013} C_VEL
LIN {X 0,Y 118.742,Z 549.473,A -85,B 0,C 180,E1 -25442.601,E2 -25442.601} C_VEL
LIN {X 0,Y 118.715,Z 547.688,A -85,B 0,C 180,E1 -25449.194,E2 -25449.194} C_VEL
LIN {X 0,Y 119.525,Z 544.964,A -85,B 0,C 180,E1 -25454.657,E2 -25454.657} C_VEL
LIN {X 0,Y 121.134,Z 540.603,A -85,B 0,C 180,E1 -25460.514,E2 -25460.514} C_VEL
LIN {X 0,Y 123.002,Z 536.061,A -85,B 0,C 180,E1 -25465.084,E2 -25465.084} C_VEL
LIN {X 0,Y 125.295,Z 530.861,A -85,B 0,C 180,E1 -25469.197,E2 -25469.197} C_VEL
LIN {X 0,Y 128.134,Z 524.548,A -85,B 0,C 180,E1 -25473.145,E2 -25473.145} C_VEL
LIN {X 0,Y 131.519,Z 516.876,A -85,B 0,C 180,E1 -25476.906,E2 -25476.906} C_VEL
LIN {X 0,Y 135.039,Z 508.281,A -85,B 0,C 180,E1 -25480.225,E2 -25480.225} C_VEL
LIN {X 0,Y 138.391,Z 499.688,A -85,B 0,C 180,E1 -25482.837,E2 -25482.837} C_VEL
LIN {X 0,Y 141.585,Z 490.337,A -85,B 0,C 180,E1 -25485.106,E2 -25485.106} C_VEL
LIN {X 0,Y 144.464,Z 480.592,A -85,B 0,C 180,E1 -25486.972,E2 -25486.972} C_VEL
LIN {X 0,Y 146.975,Z 470.506,A -85,B 0,C 180,E1 -25488.469,E2 -25488.469} C_VEL
LIN {X 0,Y 149.11,Z 459.149,A -85,B 0,C 180,E1 -25489.742,E2 -25489.742} C_VEL
LIN {X 0,Y 150.799,Z 447.677,A -85,B 0,C 180,E1 -25490.595,E2 -25490.595} C_VEL
LIN {X 0,Y 152.431,Z 429.064,A -85,B 0,C 180,E1 -25491.451,E2 -25491.451} C_VEL
LIN {X 0,Y 154.203,Z 403.46,A -85,B 0,C 180,E1 -25492.54,E2 -25492.54} C_VEL
LIN {X 0,Y 150.39,Z 393.224,A -85,B 0,C 180,E1 -25494.423,E2 -25494.423} C_VEL
LIN {X 0,Y 146.28,Z 384.899,A -85,B 0,C 180,E1 -25496.438,E2 -25496.438} C_VEL
LIN {X 0,Y 140.476,Z 374.913,A -85,B 0,C 180,E1 -25499.453,E2 -25499.453} C_VEL
LIN {X 0,Y 134.985,Z 366.26,A -85,B 0,C 180,E1 -25502.612,E2 -25502.612} C_VEL
LIN {X 0,Y 131.321,Z 361.218,A -85,B 0,C 180,E1 -25504.911,E2 -25504.911} C_VEL
LIN {X 0,Y 129.024,Z 357.902,A -85,B 0,C 180,E1 -25506.495,E2 -25506.495} C_VEL
LIN {X 0,Y 126.609,Z 355.122,A -85,B 0,C 180,E1 -25508.189,E2 -25508.189} C_VEL
LIN {X 0,Y 125.578,Z 353.15,A -85,B 0,C 180,E1 -25509.026,E2 -25509.026} C_VEL
LIN {X 0,Y 123.227,Z 351.059,A -85,B 0,C 180,E1 -25510.795,E2 -25510.795} C_VEL
LIN {X 0,Y 121.982,Z 348.607,A -85,B 0,C 180,E1 -25512.172,E2 -25512.172} C_VEL
LIN {X 0,Y 121.839,Z 347.871,A -85,B 0,C 180,E1 -25513.139,E2 -25513.139} C_VEL
LIN {X 0,Y 121.874,Z 347.767,A -85,B 0,C 180,E1 -25518.561,E2 -25518.561} C_VEL
LIN {X 0,Y 121.934,Z 347.792,A -85,B 0,C 180,E1 -25524.803,E2 -25524.803} C_VEL
LIN {X 0,Y 121.93,Z 347.743,A -85,B 0,C 180,E1 -25529.837,E2 -25529.837} C_VEL
LIN {X 0,Y 121.967,Z 347.792,A -85,B 0,C 180,E1 -25536.211,E2 -25536.211} C_VEL
LIN {X 0,Y 121.994,Z 347.737,A -85,B 0,C 180,E1 -25539.777,E2 -25539.777} C_VEL
LIN {X 0,Y 122.19,Z 347.755,A -85,B 0,C 180,E1 -25546.698,E2 -25546.698} C_VEL
LIN {X 0,Y 122.393,Z 347.706,A -85,B 0,C 180,E1 -25550.08,E2 -25550.08} C_VEL
LIN {X 0,Y 122.561,Z 347.678,A -85,B 0,C 180,E1 -25556.712,E2 -25556.712} C_VEL
LIN {X 0,Y 123.023,Z 347.656,A -85,B 0,C 180,E1 -25559.999,E2 -25559.999} C_VEL
LIN {X 0,Y 122.412,Z 347.688,A -85,B 0,C 180,E1 -25566.593,E2 -25566.593} C_VEL
LIN {X 0,Y 122.397,Z 347.738,A -85,B 0,C 180,E1 -25569.918,E2 -25569.918} C_VEL
LIN {X 0,Y 122.187,Z 347.727,A -85,B 0,C 180,E1 -25573.301,E2 -25573.301} C_VEL
LIN {X 0,Y 121.99,Z 347.784,A -85,B 0,C 180,E1 -25580.222,E2 -25580.222} C_VEL
LIN {X 0,Y 122.008,Z 347.956,A -85,B 0,C 180,E1 -25583.038,E2 -25583.038} C_VEL
LIN {X 0,Y 122.225,Z 349.133,A -85,B 0,C 180,E1 -25584.072,E2 -25584.072} C_VEL
LIN {X 0,Y 123.843,Z 351.797,A -85,B 0,C 180,E1 -25585.526,E2 -25585.526} C_VEL
LIN {X 0,Y 125.901,Z 353.531,A -85,B 0,C 180,E1 -25587.038,E2 -25587.038} C_VEL
LIN {X 0,Y 127.953,Z 356.862,A -85,B 0,C 180,E1 -25588.61,E2 -25588.61} C_VEL
LIN {X 0,Y 129.645,Z 358.682,A -85,B 0,C 180,E1 -25589.758,E2 -25589.758} C_VEL
LIN {X 0,Y 133.686,Z 364.759,A -85,B 0,C 180,E1 -25592.449,E2 -25592.449} C_VEL
LIN {X 0,Y 137.781,Z 370.74,A -85,B 0,C 180,E1 -25594.879,E2 -25594.879} C_VEL
LIN {X 0,Y 143.017,Z 379.566,A -85,B 0,C 180,E1 -25597.754,E2 -25597.754} C_VEL
LIN {X 0,Y 148.152,Z 391.102,A -85,B 0,C 180,E1 -25600.493,E2 -25600.493} C_VEL
LIN {X 0,Y 153.06,Z 404.403,A -85,B 0,C 180,E1 -25602.993,E2 -25602.993} C_VEL
LIN {X 0,Y 153.974,Z 407.075,A -85,B 0,C 180,E1 -25603.444,E2 -25603.444} C_VEL
LIN {X 0,Y 153.019,Z 421.84,A -85,B 0,C 180,E1 -25604.091,E2 -25604.091} C_VEL
LIN {X 0,Y 150.86,Z 449.267,A -85,B 0,C 180,E1 -25605.308,E2 -25605.308} C_VEL
LIN {X 0,Y 149.708,Z 458.503,A -85,B 0,C 180,E1 -25605.943,E2 -25605.943} C_VEL
LIN {X 0,Y 147.885,Z 468.73,A -85,B 0,C 180,E1 -25606.909,E2 -25606.909} C_VEL
LIN {X 0,Y 145.754,Z 477.783,A -85,B 0,C 180,E1 -25608.007,E2 -25608.007} C_VEL
LIN {X 0,Y 142.931,Z 488.502,A -85,B 0,C 180,E1 -25609.807,E2 -25609.807} C_VEL
LIN {X 0,Y 140.053,Z 497.251,A -85,B 0,C 180,E1 -25611.611,E2 -25611.611} C_VEL
LIN {X 0,Y 136.545,Z 506.84,A -85,B 0,C 180,E1 -25614.163,E2 -25614.163} C_VEL
LIN {X 0,Y 132.998,Z 515.745,A -85,B 0,C 180,E1 -25617.204,E2 -25617.204} C_VEL
LIN {X 0,Y 129.496,Z 523.919,A -85,B 0,C 180,E1 -25620.761,E2 -25620.761} C_VEL
LIN {X 0,Y 126.472,Z 530.708,A -85,B 0,C 180,E1 -25624.49,E2 -25624.49} C_VEL
LIN {X 0,Y 123.963,Z 536.366,A -85,B 0,C 180,E1 -25628.376,E2 -25628.376} C_VEL
LIN {X 0,Y 121.669,Z 541.839,A -85,B 0,C 180,E1 -25633.213,E2 -25633.213} C_VEL
LIN {X 0,Y 120.186,Z 546.111,A -85,B 0,C 180,E1 -25638.19,E2 -25638.19} C_VEL
LIN {X 0,Y 119.38,Z 549.296,A -85,B 0,C 180,E1 -25643.238,E2 -25643.238} C_VEL
LIN {X 0,Y 119.154,Z 550.915,A -85,B 0,C 180,E1 -25646.618,E2 -25646.618} C_VEL
LIN {X 0,Y 119.23,Z 551.963,A -85,B 0,C 180,E1 -25650,E2 -25650} C_VEL
LIN {X 0,Y 119.219,Z 552.737,A -85,B 0,C 180,E1 -25653.379,E2 -25653.379} C_VEL
LIN {X 0,Y 119.406,Z 553.034,A -85,B 0,C 180,E1 -25656.76,E2 -25656.76} C_VEL
LIN {X 0,Y 120.736,Z 552.565,A -85,B 0,C 180,E1 -25663.464,E2 -25663.464} C_VEL
LIN {X 0,Y 123.409,Z 550.405,A -85,B 0,C 180,E1 -25669.98,E2 -25669.98} C_VEL
LIN {X 0,Y 126.494,Z 547.786,A -85,B 0,C 180,E1 -25674.626,E2 -25674.626} C_VEL
LIN {X 0,Y 130.461,Z 544.179,A -85,B 0,C 180,E1 -25679.001,E2 -25679.001} C_VEL
LIN {X 0,Y 135.637,Z 538.635,A -85,B 0,C 180,E1 -25683.786,E2 -25683.786} C_VEL
LIN {X 0,Y 138.168,Z 535.792,A -85,B 0,C 180,E1 -25685.742,E2 -25685.742} C_VEL
LIN {X 0,Y 140.262,Z 532.909,A -85,B 0,C 180,E1 -25687.685,E2 -25687.685} C_VEL
LIN {X 0,Y 142.488,Z 527.86,A -85,B 0,C 180,E1 -25691.027,E2 -25691.027} C_VEL
LIN {X 0,Y 144.913,Z 522.194,A -85,B 0,C 180,E1 -25694.107,E2 -25694.107} C_VEL
LIN {X 0,Y 147.218,Z 518.292,A -85,B 0,C 180,E1 -25695.595,E2 -25695.595} C_VEL
LIN {X 0,Y 152.071,Z 510.995,A -85,B 0,C 180,E1 -25697.684,E2 -25697.684} C_VEL
LIN {X 0,Y 157.017,Z 502.631,A -85,B 0,C 180,E1 -25699.544,E2 -25699.544} C_VEL
LIN {X 0,Y 162.093,Z 492.477,A -85,B 0,C 180,E1 -25701.301,E2 -25701.301} C_VEL
LIN {X 0,Y 166.007,Z 483.229,A -85,B 0,C 180,E1 -25702.541,E2 -25702.541} C_VEL
LIN {X 0,Y 169.567,Z 472.984,A -85,B 0,C 180,E1 -25703.594,E2 -25703.594} C_VEL
LIN {X 0,Y 172.639,Z 461.72,A -85,B 0,C 180,E1 -25704.419,E2 -25704.419} C_VEL
LIN {X 0,Y 174.795,Z 450.602,A -85,B 0,C 180,E1 -25705.005,E2 -25705.005} C_VEL
LIN {X 0,Y 176.898,Z 431.944,A -85,B 0,C 180,E1 -25705.693,E2 -25705.693} C_VEL
LIN {X 0,Y 177.38,Z 426.697,A -85,B 0,C 180,E1 -25705.888,E2 -25705.888} C_VEL
LIN {X 0,Y 174.8,Z 419.357,A -85,B 0,C 180,E1 -25708.572,E2 -25708.572} C_VEL
LIN {X 0,Y 172.189,Z 412.927,A -85,B 0,C 180,E1 -25711.66,E2 -25711.66} C_VEL
LIN {X 0,Y 170.879,Z 410.187,A -85,B 0,C 180,E1 -25713.437,E2 -25713.437} C_VEL
LIN {X 0,Y 169.072,Z 406.888,A -85,B 0,C 180,E1 -25716.245,E2 -25716.245} C_VEL
LIN {X 0,Y 167.167,Z 403.413,A -85,B 0,C 180,E1 -25720.347,E2 -25720.347} C_VEL
LIN {X 0,Y 166.664,Z 402.733,A -85,B 0,C 180,E1 -25721.763,E2 -25721.763} C_VEL
LIN {X 0,Y 165.669,Z 401.396,A -85,B 0,C 180,E1 -25727.755,E2 -25727.755} C_VEL
LIN {X 0,Y 165.956,Z 401.668,A -85,B 0,C 180,E1 -25731.4,E2 -25731.4} C_VEL
LIN {X 0,Y 167.409,Z 403.152,A -85,B 0,C 180,E1 -25736.339,E2 -25736.339} C_VEL
LIN {X 0,Y 169.111,Z 406.573,A -85,B 0,C 180,E1 -25740.001,E2 -25740.001} C_VEL
LIN {X 0,Y 169.926,Z 407.889,A -85,B 0,C 180,E1 -25741.306,E2 -25741.306} C_VEL
LIN {X 0,Y 171.881,Z 411.734,A -85,B 0,C 180,E1 -25744.122,E2 -25744.122} C_VEL
LIN {X 0,Y 174.5,Z 416.719,A -85,B 0,C 180,E1 -25747.123,E2 -25747.123} C_VEL
LIN {X 0,Y 176.437,Z 421.061,A -85,B 0,C 180,E1 -25749.127,E2 -25749.127} C_VEL
LIN {X 0,Y 177.636,Z 424.221,A -85,B 0,C 180,E1 -25750.289,E2 -25750.289} C_VEL
LIN {X 0,Y 175.136,Z 446.828,A -85,B 0,C 180,E1 -25751.047,E2 -25751.047} C_VEL
LIN {X 0,Y 173.492,Z 456.316,A -85,B 0,C 180,E1 -25751.531,E2 -25751.531} C_VEL
LIN {X 0,Y 171.377,Z 465.271,A -85,B 0,C 180,E1 -25752.125,E2 -25752.125} C_VEL
LIN {X 0,Y 168.207,Z 475.737,A -85,B 0,C 180,E1 -25753.085,E2 -25753.085} C_VEL
LIN {X 0,Y 164.485,Z 485.593,A -85,B 0,C 180,E1 -25754.27,E2 -25754.27} C_VEL
LIN {X 0,Y 159.82,Z 495.73,A -85,B 0,C 180,E1 -25755.859,E2 -25755.859} C_VEL
LIN {X 0,Y 154.919,Z 504.779,A -85,B 0,C 180,E1 -25757.697,E2 -25757.697} C_VEL
LIN {X 0,Y 149.525,Z 513.36,A -85,B 0,C 180,E1 -25759.942,E2 -25759.942} C_VEL
LIN {X 0,Y 144.385,Z 520.573,A -85,B 0,C 180,E1 -25762.358,E2 -25762.358} C_VEL
LIN {X 0,Y 138.301,Z 528.006,A -85,B 0,C 180,E1 -25765.579,E2 -25765.579} C_VEL
LIN {X 0,Y 134.212,Z 532.641,A -85,B 0,C 180,E1 -25768.119,E2 -25768.119} C_VEL
LIN {X 0,Y 128.679,Z 538.195,A -85,B 0,C 180,E1 -25772.165,E2 -25772.165} C_VEL
LIN {X 0,Y 123.36,Z 542.967,A -85,B 0,C 180,E1 -25777.099,E2 -25777.099} C_VEL
LIN {X 0,Y 120.34,Z 545.503,A -85,B 0,C 180,E1 -25780.605,E2 -25780.605} C_VEL
LIN {X 0,Y 116.48,Z 548.215,A -85,B 0,C 180,E1 -25786.39,E2 -25786.39} C_VEL
LIN {X 0,Y 113.979,Z 549.604,A -85,B 0,C 180,E1 -25791.932,E2 -25791.932} C_VEL
LIN {X 0,Y 112.763,Z 549.935,A -85,B 0,C 180,E1 -25795.88,E2 -25795.88} C_VEL
LIN {X 0,Y 111.569,Z 549.227,A -85,B 0,C 180,E1 -25803.836,E2 -25803.836} C_VEL
LIN {X 0,Y 111.531,Z 548.155,A -85,B 0,C 180,E1 -25807.785,E2 -25807.785} C_VEL
LIN {X 0,Y 111.906,Z 546.54,A -85,B 0,C 180,E1 -25811.699,E2 -25811.699} C_VEL
LIN {X 0,Y 113.058,Z 543.302,A -85,B 0,C 180,E1 -25817.434,E2 -25817.434} C_VEL
LIN {X 0,Y 114.403,Z 539.967,A -85,B 0,C 180,E1 -25821.795,E2 -25821.795} C_VEL
LIN {X 0,Y 115.591,Z 537.295,A -85,B 0,C 180,E1 -25824.768,E2 -25824.768} C_VEL
LIN {X 0,Y 118.395,Z 531.158,A -85,B 0,C 180,E1 -25830,E2 -25830} C_VEL
LIN {X 0,Y 121.378,Z 524.883,A -85,B 0,C 180,E1 -25834.151,E2 -25834.151} C_VEL
LIN {X 0,Y 124.943,Z 517.252,A -85,B 0,C 180,E1 -25838.084,E2 -25838.084} C_VEL
LIN {X 0,Y 128.241,Z 509.659,A -85,B 0,C 180,E1 -25841.219,E2 -25841.219} C_VEL
LIN {X 0,Y 132.115,Z 500.189,A -85,B 0,C 180,E1 -25844.243,E2 -25844.243} C_VEL
LIN {X 0,Y 135.457,Z 490.919,A -85,B 0,C 180,E1 -25846.581,E2 -25846.581} C_VEL
LIN {X 0,Y 138.449,Z 481.297,A -85,B 0,C 180,E1 -25848.498,E2 -25848.498} C_VEL
LIN {X 0,Y 141.324,Z 470.149,A -85,B 0,C 180,E1 -25850.182,E2 -25850.182} C_VEL
LIN {X 0,Y 143.478,Z 459.138,A -85,B 0,C 180,E1 -25851.433,E2 -25851.433} C_VEL
LIN {X 0,Y 145.174,Z 448.212,A -85,B 0,C 180,E1 -25852.263,E2 -25852.263} C_VEL
LIN {X 0,Y 146.89,Z 429.459,A -85,B 0,C 180,E1 -25853.147,E2 -25853.147} C_VEL
LIN {X 0,Y 148.707,Z 405.282,A -85,B 0,C 180,E1 -25854.174,E2 -25854.174} C_VEL
LIN {X 0,Y 144.557,Z 394.589,A -85,B 0,C 180,E1 -25856.383,E2 -25856.383} C_VEL
LIN {X 0,Y 139.216,Z 384.511,A -85,B 0,C 180,E1 -25859.234,E2 -25859.234} C_VEL
LIN {X 0,Y 133.484,Z 374.913,A -85,B 0,C 180,E1 -25862.603,E2 -25862.603} C_VEL
LIN {X 0,Y 128.396,Z 367.265,A -85,B 0,C 180,E1 -25865.954,E2 -25865.954} C_VEL
LIN {X 0,Y 125.84,Z 363.711,A -85,B 0,C 180,E1 -25867.794,E2 -25867.794} C_VEL
LIN {X 0,Y 123.167,Z 360.187,A -85,B 0,C 180,E1 -25869.85,E2 -25869.85} C_VEL
LIN {X 0,Y 122.337,Z 358.969,A -85,B 0,C 180,E1 -25870.541,E2 -25870.541} C_VEL
LIN {X 0,Y 119.863,Z 356.105,A -85,B 0,C 180,E1 -25872.649,E2 -25872.649} C_VEL
LIN {X 0,Y 118.744,Z 354.202,A -85,B 0,C 180,E1 -25873.748,E2 -25873.748} C_VEL
LIN {X 0,Y 116.276,Z 352.213,A -85,B 0,C 180,E1 -25876.063,E2 -25876.063} C_VEL
LIN {X 0,Y 114.998,Z 349.634,A -85,B 0,C 180,E1 -25877.758,E2 -25877.758} C_VEL
LIN {X 0,Y 114.839,Z 348.716,A -85,B 0,C 180,E1 -25879.15,E2 -25879.15} C_VEL
LIN {X 0,Y 114.799,Z 348.649,A -85,B 0,C 180,E1 -25882.738,E2 -25882.738} C_VEL
LIN {X 0,Y 114.863,Z 348.627,A -85,B 0,C 180,E1 -25888.938,E2 -25888.938} C_VEL
LIN {X 0,Y 114.931,Z 348.667,A -85,B 0,C 180,E1 -25896.527,E2 -25896.527} C_VEL
LIN {X 0,Y 114.971,Z 348.601,A -85,B 0,C 180,E1 -25902.202,E2 -25902.202} C_VEL
LIN {X 0,Y 115.307,Z 348.596,A -85,B 0,C 180,E1 -25909.463,E2 -25909.463} C_VEL
LIN {X 0,Y 115.487,Z 348.554,A -85,B 0,C 180,E1 -25916.51,E2 -25916.51} C_VEL
LIN {X 0,Y 115.975,Z 348.532,A -85,B 0,C 180,E1 -25919.999,E2 -25919.999} C_VEL
LIN {X 0,Y 115.354,Z 348.569,A -85,B 0,C 180,E1 -25926.998,E2 -25926.998} C_VEL
LIN {X 0,Y 115.204,Z 348.602,A -85,B 0,C 180,E1 -25932.557,E2 -25932.557} C_VEL
LIN {X 0,Y 115.023,Z 348.89,A -85,B 0,C 180,E1 -25937.329,E2 -25937.329} C_VEL
LIN {X 0,Y 115.283,Z 350.112,A -85,B 0,C 180,E1 -25938.55,E2 -25938.55} C_VEL
LIN {X 0,Y 116.782,Z 352.609,A -85,B 0,C 180,E1 -25940.244,E2 -25940.244} C_VEL
LIN {X 0,Y 119.108,Z 354.482,A -85,B 0,C 180,E1 -25942.401,E2 -25942.401} C_VEL
LIN {X 0,Y 121.016,Z 357.697,A -85,B 0,C 180,E1 -25944.213,E2 -25944.213} C_VEL
LIN {X 0,Y 123.015,Z 359.735,A -85,B 0,C 180,E1 -25945.824,E2 -25945.824} C_VEL
LIN {X 0,Y 125.697,Z 363.488,A -85,B 0,C 180,E1 -25947.921,E2 -25947.921} C_VEL
LIN {X 0,Y 129.472,Z 368.952,A -85,B 0,C 180,E1 -25950.623,E2 -25950.623} C_VEL
LIN {X 0,Y 134.273,Z 376.326,A -85,B 0,C 180,E1 -25953.722,E2 -25953.722} C_VEL
LIN {X 0,Y 138.946,Z 384.52,A -85,B 0,C 180,E1 -25956.477,E2 -25956.477} C_VEL
LIN {X 0,Y 143.797,Z 395.852,A -85,B 0,C 180,E1 -25959.25,E2 -25959.25} C_VEL
LIN {X 0,Y 148.368,Z 408.85,A -85,B 0,C 180,E1 -25961.779,E2 -25961.779} C_VEL
LIN {X 0,Y 148.098,Z 415.286,A -85,B 0,C 180,E1 -25962.123,E2 -25962.123} C_VEL
LIN {X 0,Y 145.348,Z 448.622,A -85,B 0,C 180,E1 -25963.581,E2 -25963.581} C_VEL
LIN {X 0,Y 144.102,Z 458.304,A -85,B 0,C 180,E1 -25964.248,E2 -25964.248} C_VEL
LIN {X 0,Y 142.207,Z 468.558,A -85,B 0,C 180,E1 -25965.231,E2 -25965.231} C_VEL
LIN {X 0,Y 139.992,Z 477.626,A -85,B 0,C 180,E1 -25966.346,E2 -25966.346} C_VEL
LIN {X 0,Y 137.042,Z 488.357,A -85,B 0,C 180,E1 -25968.188,E2 -25968.188} C_VEL
LIN {X 0,Y 134.044,Z 497.115,A -85,B 0,C 180,E1 -25970.038,E2 -25970.038} C_VEL
LIN {X 0,Y 130.375,Z 506.711,A -85,B 0,C 180,E1 -25972.667,E2 -25972.667} C_VEL
LIN {X 0,Y 127.042,Z 514.76,A -85,B 0,C 180,E1 -25975.456,E2 -25975.456} C_VEL
LIN {X 0,Y 123.248,Z 523.074,A -85,B 0,C 180,E1 -25979.122,E2 -25979.122} C_VEL
LIN {X 0,Y 120.059,Z 529.999,A -85,B 0,C 180,E1 -25983.02,E2 -25983.02} C_VEL
LIN {X 0,Y 117.376,Z 535.772,A -85,B 0,C 180,E1 -25987.095,E2 -25987.095} C_VEL
LIN {X 0,Y 114.834,Z 541.344,A -85,B 0,C 180,E1 -25992.181,E2 -25992.181} C_VEL
LIN {X 0,Y 113.222,Z 545.714,A -85,B 0,C 180,E1 -25997.452,E2 -25997.452} C_VEL
LIN {X 0,Y 112.312,Z 548.987,A -85,B 0,C 180,E1 -26002.81,E2 -26002.81} C_VEL
LIN {X 0,Y 112.086,Z 550.609,A -85,B 0,C 180,E1 -26006.405,E2 -26006.405} C_VEL
LIN {X 0,Y 112.135,Z 551.739,A -85,B 0,C 180,E1 -26010,E2 -26010} C_VEL
LIN {X 0,Y 112.13,Z 552.595,A -85,B 0,C 180,E1 -26013.593,E2 -26013.593} C_VEL
LIN {X 0,Y 112.902,Z 552.871,A -85,B 0,C 180,E1 -26020.763,E2 -26020.763} C_VEL
LIN {X 0,Y 113.814,Z 552.528,A -85,B 0,C 180,E1 -26024.3,E2 -26024.3} C_VEL
LIN {X 0,Y 116.734,Z 550.521,A -85,B 0,C 180,E1 -26031.176,E2 -26031.176} C_VEL
LIN {X 0,Y 120.083,Z 548.001,A -85,B 0,C 180,E1 -26036.036,E2 -26036.036} C_VEL
LIN {X 0,Y 124.294,Z 544.493,A -85,B 0,C 180,E1 -26040.59,E2 -26040.59} C_VEL
LIN {X 0,Y 129.55,Z 539.348,A -85,B 0,C 180,E1 -26045.321,E2 -26045.321} C_VEL
LIN {X 0,Y 135.442,Z 533.015,A -85,B 0,C 180,E1 -26049.467,E2 -26049.467} C_VEL
LIN {X 0,Y 140.625,Z 526.974,A -85,B 0,C 180,E1 -26052.43,E2 -26052.43} C_VEL
LIN {X 0,Y 146.242,Z 519.731,A -85,B 0,C 180,E1 -26055.141,E2 -26055.141} C_VEL
LIN {X 0,Y 147.218,Z 518.292,A -85,B 0,C 180,E1 -26055.595,E2 -26055.595} C_VEL
LIN {X 0,Y 149.526,Z 514.414,A -85,B 0,C 180,E1 -26057.004,E2 -26057.004} C_VEL
LIN {X 0,Y 153.169,Z 504.926,A -85,B 0,C 180,E1 -26060.635,E2 -26060.635} C_VEL
LIN {X 0,Y 155.421,Z 499.009,A -85,B 0,C 180,E1 -26062.374,E2 -26062.374} C_VEL
LIN {X 0,Y 156.997,Z 495.817,A -85,B 0,C 180,E1 -26063.023,E2 -26063.023} C_VEL
LIN {X 0,Y 162.537,Z 483.505,A -85,B 0,C 180,E1 -26064.7,E2 -26064.7} C_VEL
LIN {X 0,Y 166.331,Z 473.015,A -85,B 0,C 180,E1 -26065.749,E2 -26065.749} C_VEL
LIN {X 0,Y 169.565,Z 461.55,A -85,B 0,C 180,E1 -26066.562,E2 -26066.562} C_VEL
LIN {X 0,Y 171.782,Z 450.439,A -85,B 0,C 180,E1 -26067.136,E2 -26067.136} C_VEL
LIN {X 0,Y 173.931,Z 432.243,A -85,B 0,C 180,E1 -26067.794,E2 -26067.794} C_VEL
LIN {X 0,Y 174.061,Z 429.644,A -85,B 0,C 180,E1 -26067.985,E2 -26067.985} C_VEL
LIN {X 0,Y 171.619,Z 422.371,A -85,B 0,C 180,E1 -26070.939,E2 -26070.939} C_VEL
LIN {X 0,Y 169.469,Z 416.977,A -85,B 0,C 180,E1 -26073.973,E2 -26073.973} C_VEL
LIN {X 0,Y 167.72,Z 413.66,A -85,B 0,C 180,E1 -26076.848,E2 -26076.848} C_VEL
LIN {X 0,Y 165.92,Z 409.964,A -85,B 0,C 180,E1 -26081.185,E2 -26081.185} C_VEL
LIN {X 0,Y 164.733,Z 408.436,A -85,B 0,C 180,E1 -26087.684,E2 -26087.684} C_VEL
LIN {X 0,Y 165.005,Z 408.711,A -85,B 0,C 180,E1 -26091.35,E2 -26091.35} C_VEL
LIN {X 0,Y 166.214,Z 409.988,A -85,B 0,C 180,E1 -26095.757,E2 -26095.757} C_VEL
LIN {X 0,Y 167.994,Z 413.572,A -85,B 0,C 180,E1 -26099.782,E2 -26099.782} C_VEL
LIN {X 0,Y 170.062,Z 417.869,A -85,B 0,C 180,E1 -26103.092,E2 -26103.092} C_VEL
LIN {X 0,Y 172.664,Z 423.318,A -85,B 0,C 180,E1 -26106.368,E2 -26106.368} C_VEL
LIN {X 0,Y 174.111,Z 426.84,A -85,B 0,C 180,E1 -26107.985,E2 -26107.985} C_VEL
LIN {X 0,Y 174.382,Z 427.596,A -85,B 0,C 180,E1 -26108.283,E2 -26108.283} C_VEL
LIN {X 0,Y 172.082,Z 447.276,A -85,B 0,C 180,E1 -26108.943,E2 -26108.943} C_VEL
LIN {X 0,Y 170.251,Z 457.155,A -85,B 0,C 180,E1 -26109.435,E2 -26109.435} C_VEL
LIN {X 0,Y 167.91,Z 466.447,A -85,B 0,C 180,E1 -26110.062,E2 -26110.062} C_VEL
LIN {X 0,Y 164.664,Z 476.571,A -85,B 0,C 180,E1 -26110.991,E2 -26110.991} C_VEL
LIN {X 0,Y 160.769,Z 486.364,A -85,B 0,C 180,E1 -26112.162,E2 -26112.162} C_VEL
LIN {X 0,Y 156.353,Z 495.618,A -85,B 0,C 180,E1 -26113.583,E2 -26113.583} C_VEL
LIN {X 0,Y 151.421,Z 504.408,A -85,B 0,C 180,E1 -26115.307,E2 -26115.307} C_VEL
LIN {X 0,Y 145.603,Z 513.299,A -85,B 0,C 180,E1 -26117.581,E2 -26117.581} C_VEL
LIN {X 0,Y 139.719,Z 521.123,A -85,B 0,C 180,E1 -26120.204,E2 -26120.204} C_VEL
LIN {X 0,Y 133.791,Z 527.982,A -85,B 0,C 180,E1 -26123.181,E2 -26123.181} C_VEL
LIN {X 0,Y 128.08,Z 533.89,A -85,B 0,C 180,E1 -26126.6,E2 -26126.6} C_VEL
LIN {X 0,Y 122.502,Z 539.031,A -85,B 0,C 180,E1 -26130.622,E2 -26130.622} C_VEL
LIN {X 0,Y 118.665,Z 542.335,A -85,B 0,C 180,E1 -26133.988,E2 -26133.988} C_VEL
LIN {X 0,Y 115.211,Z 544.929,A -85,B 0,C 180,E1 -26137.591,E2 -26137.591} C_VEL
LIN {X 0,Y 110.142,Z 548.302,A -85,B 0,C 180,E1 -26144.58,E2 -26144.58} C_VEL
LIN {X 0,Y 107.775,Z 549.521,A -85,B 0,C 180,E1 -26149.3,E2 -26149.3} C_VEL
LIN {X 0,Y 106.26,Z 549.944,A -85,B 0,C 180,E1 -26153.47,E2 -26153.47} C_VEL
LIN {X 0,Y 104.714,Z 549.709,A -85,B 0,C 180,E1 -26160.753,E2 -26160.753} C_VEL
LIN {X 0,Y 104.391,Z 548.566,A -85,B 0,C 180,E1 -26166.176,E2 -26166.176} C_VEL
LIN {X 0,Y 104.647,Z 547.153,A -85,B 0,C 180,E1 -26170.379,E2 -26170.379} C_VEL
LIN {X 0,Y 105.206,Z 545.355,A -85,B 0,C 180,E1 -26174.502,E2 -26174.502} C_VEL
LIN {X 0,Y 106.824,Z 541.432,A -85,B 0,C 180,E1 -26180.705,E2 -26180.705} C_VEL
LIN {X 0,Y 109.465,Z 535.572,A -85,B 0,C 180,E1 -26187.24,E2 -26187.24} C_VEL
LIN {X 0,Y 111.86,Z 530.744,A -85,B 0,C 180,E1 -26191.417,E2 -26191.417} C_VEL
LIN {X 0,Y 115.385,Z 523.724,A -85,B 0,C 180,E1 -26196.119,E2 -26196.119} C_VEL
LIN {X 0,Y 118.434,Z 517.625,A -85,B 0,C 180,E1 -26199.392,E2 -26199.392} C_VEL
LIN {X 0,Y 122.594,Z 508.387,A -85,B 0,C 180,E1 -26203.257,E2 -26203.257} C_VEL
LIN {X 0,Y 126.45,Z 499.394,A -85,B 0,C 180,E1 -26206.135,E2 -26206.135} C_VEL
LIN {X 0,Y 129.934,Z 489.951,A -85,B 0,C 180,E1 -26208.529,E2 -26208.529} C_VEL
LIN {X 0,Y 133.099,Z 480.06,A -85,B 0,C 180,E1 -26210.477,E2 -26210.477} C_VEL
LIN {X 0,Y 135.869,Z 469.562,A -85,B 0,C 180,E1 -26212.062,E2 -26212.062} C_VEL
LIN {X 0,Y 138.094,Z 458.409,A -85,B 0,C 180,E1 -26213.327,E2 -26213.327} C_VEL
LIN {X 0,Y 139.746,Z 448.067,A -85,B 0,C 180,E1 -26214.108,E2 -26214.108} C_VEL
LIN {X 0,Y 141.431,Z 430.514,A -85,B 0,C 180,E1 -26214.948,E2 -26214.948} C_VEL
LIN {X 0,Y 143.283,Z 407.276,A -85,B 0,C 180,E1 -26215.943,E2 -26215.943} C_VEL
LIN {X 0,Y 139.785,Z 398.183,A -85,B 0,C 180,E1 -26217.954,E2 -26217.954} C_VEL
LIN {X 0,Y 134.866,Z 388.793,A -85,B 0,C 180,E1 -26220.783,E2 -26220.783} C_VEL
LIN {X 0,Y 129.531,Z 379.656,A -85,B 0,C 180,E1 -26224.19,E2 -26224.19} C_VEL
LIN {X 0,Y 124.634,Z 372.121,A -85,B 0,C 180,E1 -26227.676,E2 -26227.676} C_VEL
LIN {X 0,Y 122.79,Z 369.484,A -85,B 0,C 180,E1 -26229.113,E2 -26229.113} C_VEL
LIN {X 0,Y 119.98,Z 365.507,A -85,B 0,C 180,E1 -26231.471,E2 -26231.471} C_VEL
LIN {X 0,Y 116.92,Z 361.597,A -85,B 0,C 180,E1 -26234.3,E2 -26234.3} C_VEL
LIN {X 0,Y 116.217,Z 360.495,A -85,B 0,C 180,E1 -26235.026,E2 -26235.026} C_VEL
LIN {X 0,Y 113.866,Z 358.311,A -85,B 0,C 180,E1 -26237.402,E2 -26237.402} C_VEL
LIN {X 0,Y 112.209,Z 355.297,A -85,B 0,C 180,E1 -26239.469,E2 -26239.469} C_VEL
LIN {X 0,Y 109.513,Z 353.397,A -85,B 0,C 180,E1 -26242.826,E2 -26242.826} C_VEL
LIN {X 0,Y 107.994,Z 350.739,A -85,B 0,C 180,E1 -26245.486,E2 -26245.486} C_VEL
LIN {X 0,Y 107.788,Z 349.622,A -85,B 0,C 180,E1 -26247.515,E2 -26247.515} C_VEL
LIN {X 0,Y 107.844,Z 349.549,A -85,B 0,C 180,E1 -26255.834,E2 -26255.834} C_VEL
LIN {X 0,Y 107.87,Z 349.486,A -85,B 0,C 180,E1 -26260.987,E2 -26260.987} C_VEL
LIN {X 0,Y 108.226,Z 349.488,A -85,B 0,C 180,E1 -26268.765,E2 -26268.765} C_VEL
LIN {X 0,Y 108.288,Z 349.434,A -85,B 0,C 180,E1 -26272.541,E2 -26272.541} C_VEL
LIN {X 0,Y 108.9,Z 349.41,A -85,B 0,C 180,E1 -26279.999,E2 -26279.999} C_VEL
LIN {X 0,Y 108.266,Z 349.636,A -85,B 0,C 180,E1 -26289.221,E2 -26289.221} C_VEL
LIN {X 0,Y 108.535,Z 350.87,A -85,B 0,C 180,E1 -26291.2,E2 -26291.2} C_VEL
LIN {X 0,Y 110.149,Z 353.689,A -85,B 0,C 180,E1 -26293.821,E2 -26293.821} C_VEL
LIN {X 0,Y 112.577,Z 355.634,A -85,B 0,C 180,E1 -26296.781,E2 -26296.781} C_VEL
LIN {X 0,Y 114.177,Z 358.517,A -85,B 0,C 180,E1 -26298.736,E2 -26298.736} C_VEL
LIN {X 0,Y 116.622,Z 360.958,A -85,B 0,C 180,E1 -26301.196,E2 -26301.196} C_VEL
LIN {X 0,Y 118.977,Z 364.416,A -85,B 0,C 180,E1 -26303.488,E2 -26303.488} C_VEL
LIN {X 0,Y 120.265,Z 365.901,A -85,B 0,C 180,E1 -26304.605,E2 -26304.605} C_VEL
LIN {X 0,Y 123.981,Z 371.222,A -85,B 0,C 180,E1 -26307.652,E2 -26307.652} C_VEL
LIN {X 0,Y 128.99,Z 378.911,A -85,B 0,C 180,E1 -26311.281,E2 -26311.281} C_VEL
LIN {X 0,Y 134.138,Z 387.735,A -85,B 0,C 180,E1 -26314.62,E2 -26314.62} C_VEL
LIN {X 0,Y 138.815,Z 398.78,A -85,B 0,C 180,E1 -26317.525,E2 -26317.525} C_VEL
LIN {X 0,Y 143.026,Z 411.014,A -85,B 0,C 180,E1 -26320.059,E2 -26320.059} C_VEL
LIN {X 0,Y 139.986,Z 447.821,A -85,B 0,C 180,E1 -26321.707,E2 -26321.707} C_VEL
LIN {X 0,Y 138.682,Z 457.872,A -85,B 0,C 180,E1 -26322.4,E2 -26322.4} C_VEL
LIN {X 0,Y 136.642,Z 468.476,A -85,B 0,C 180,E1 -26323.426,E2 -26323.426} C_VEL
LIN {X 0,Y 134.359,Z 477.469,A -85,B 0,C 180,E1 -26324.545,E2 -26324.545} C_VEL
LIN {X 0,Y 131.279,Z 488.214,A -85,B 0,C 180,E1 -26326.428,E2 -26326.428} C_VEL
LIN {X 0,Y 128.145,Z 496.979,A -85,B 0,C 180,E1 -26328.318,E2 -26328.318} C_VEL
LIN {X 0,Y 124.303,Z 506.582,A -85,B 0,C 180,E1 -26331.023,E2 -26331.023} C_VEL
LIN {X 0,Y 120.384,Z 515.499,A -85,B 0,C 180,E1 -26334.281,E2 -26334.281} C_VEL
LIN {X 0,Y 116.469,Z 523.679,A -85,B 0,C 180,E1 -26338.129,E2 -26338.129} C_VEL
LIN {X 0,Y 113.749,Z 529.291,A -85,B 0,C 180,E1 -26341.39,E2 -26341.39} C_VEL
LIN {X 0,Y 110.847,Z 535.169,A -85,B 0,C 180,E1 -26345.662,E2 -26345.662} C_VEL
LIN {X 0,Y 108.045,Z 540.85,A -85,B 0,C 180,E1 -26351.02,E2 -26351.02} C_VEL
LIN {X 0,Y 106.291,Z 545.317,A -85,B 0,C 180,E1 -26356.619,E2 -26356.619} C_VEL
LIN {X 0,Y 105.266,Z 548.679,A -85,B 0,C 180,E1 -26362.326,E2 -26362.326} C_VEL
LIN {X 0,Y 105.01,Z 550.302,A -85,B 0,C 180,E1 -26366.162,E2 -26366.162} C_VEL
LIN {X 0,Y 105.034,Z 551.516,A -85,B 0,C 180,E1 -26370,E2 -26370} C_VEL
LIN {X 0,Y 105.04,Z 552.428,A -85,B 0,C 180,E1 -26373.836,E2 -26373.836} C_VEL
LIN {X 0,Y 105.913,Z 552.814,A -85,B 0,C 180,E1 -26381.482,E2 -26381.482} C_VEL
LIN {X 0,Y 106.93,Z 552.473,A -85,B 0,C 180,E1 -26385.242,E2 -26385.242} C_VEL
LIN {X 0,Y 110.119,Z 550.642,A -85,B 0,C 180,E1 -26392.515,E2 -26392.515} C_VEL
LIN {X 0,Y 115.148,Z 547.074,A -85,B 0,C 180,E1 -26399.227,E2 -26399.227} C_VEL
LIN {X 0,Y 119.797,Z 543.321,A -85,B 0,C 180,E1 -26403.871,E2 -26403.871} C_VEL
LIN {X 0,Y 125.077,Z 538.498,A -85,B 0,C 180,E1 -26408.176,E2 -26408.176} C_VEL
LIN {X 0,Y 130.075,Z 533.597,A -85,B 0,C 180,E1 -26411.443,E2 -26411.443} C_VEL
LIN {X 0,Y 136.66,Z 526.319,A -85,B 0,C 180,E1 -26415.001,E2 -26415.001} C_VEL
LIN {X 0,Y 142.552,Z 518.977,A -85,B 0,C 180,E1 -26417.69,E2 -26417.69} C_VEL
LIN {X 0,Y 148.056,Z 511.111,A -85,B 0,C 180,E1 -26419.945,E2 -26419.945} C_VEL
LIN {X 0,Y 153.217,Z 502.783,A -85,B 0,C 180,E1 -26421.768,E2 -26421.768} C_VEL
LIN {X 0,Y 156.997,Z 495.817,A -85,B 0,C 180,E1 -26423.023,E2 -26423.023} C_VEL
LIN {X 0,Y 159.144,Z 490.998,A -85,B 0,C 180,E1 -26423.992,E2 -26423.992} C_VEL
LIN {X 0,Y 161.327,Z 482.973,A -85,B 0,C 180,E1 -26425.929,E2 -26425.929} C_VEL
LIN {X 0,Y 163.217,Z 474.569,A -85,B 0,C 180,E1 -26427.656,E2 -26427.656} C_VEL
LIN {X 0,Y 164.62,Z 469.164,A -85,B 0,C 180,E1 -26428.291,E2 -26428.291} C_VEL
LIN {X 0,Y 167.175,Z 459.707,A -85,B 0,C 180,E1 -26428.893,E2 -26428.893} C_VEL
LIN {X 0,Y 169.167,Z 449.538,A -85,B 0,C 180,E1 -26429.391,E2 -26429.391} C_VEL
LIN {X 0,Y 171.124,Z 433.136,A -85,B 0,C 180,E1 -26430.008,E2 -26430.008} C_VEL
LIN {X 0,Y 169.181,Z 427.143,A -85,B 0,C 180,E1 -26432.704,E2 -26432.704} C_VEL
LIN {X 0,Y 167.746,Z 423.237,A -85,B 0,C 180,E1 -26435.022,E2 -26435.022} C_VEL
LIN {X 0,Y 166.127,Z 419.959,A -85,B 0,C 180,E1 -26438.025,E2 -26438.025} C_VEL
LIN {X 0,Y 164.662,Z 416.754,A -85,B 0,C 180,E1 -26442.076,E2 -26442.076} C_VEL
LIN {X 0,Y 163.794,Z 415.491,A -85,B 0,C 180,E1 -26447.612,E2 -26447.612} C_VEL
LIN {X 0,Y 164.055,Z 415.748,A -85,B 0,C 180,E1 -26451.299,E2 -26451.299} C_VEL
LIN {X 0,Y 165.091,Z 416.981,A -85,B 0,C 180,E1 -26455.346,E2 -26455.346} C_VEL
LIN {X 0,Y 166.997,Z 421.115,A -85,B 0,C 180,E1 -26459.836,E2 -26459.836} C_VEL
LIN {X 0,Y 169.168,Z 425.922,A -85,B 0,C 180,E1 -26463.344,E2 -26463.344} C_VEL
LIN {X 0,Y 171.391,Z 431.117,A -85,B 0,C 180,E1 -26466.226,E2 -26466.226} C_VEL
LIN {X 0,Y 169.141,Z 448.834,A -85,B 0,C 180,E1 -26466.792,E2 -26466.792} C_VEL
LIN {X 0,Y 166.392,Z 462.025,A -85,B 0,C 180,E1 -26467.488,E2 -26467.488} C_VEL
LIN {X 0,Y 162.151,Z 475.551,A -85,B 0,C 180,E1 -26468.605,E2 -26468.605} C_VEL
LIN {X 0,Y 157.803,Z 486.189,A -85,B 0,C 180,E1 -26469.813,E2 -26469.813} C_VEL
LIN {X 0,Y 152.962,Z 495.912,A -85,B 0,C 180,E1 -26471.262,E2 -26471.262} C_VEL
LIN {X 0,Y 147.833,Z 504.659,A -85,B 0,C 180,E1 -26472.949,E2 -26472.949} C_VEL
LIN {X 0,Y 141.95,Z 513.261,A -85,B 0,C 180,E1 -26475.106,E2 -26475.106} C_VEL
LIN {X 0,Y 136.48,Z 520.304,A -85,B 0,C 180,E1 -26477.382,E2 -26477.382} C_VEL
LIN {X 0,Y 129.54,Z 527.973,A -85,B 0,C 180,E1 -26480.631,E2 -26480.631} C_VEL
LIN {X 0,Y 123.26,Z 534.092,A -85,B 0,C 180,E1 -26484.178,E2 -26484.178} C_VEL
LIN {X 0,Y 118.623,Z 538.219,A -85,B 0,C 180,E1 -26487.291,E2 -26487.291} C_VEL
LIN {X 0,Y 112.37,Z 543.018,A -85,B 0,C 180,E1 -26492.4,E2 -26492.4} C_VEL
LIN {X 0,Y 107.106,Z 546.513,A -85,B 0,C 180,E1 -26498.057,E2 -26498.057} C_VEL
LIN {X 0,Y 103.928,Z 548.389,A -85,B 0,C 180,E1 -26502.551,E2 -26502.551} C_VEL
LIN {X 0,Y 99.972,Z 549.953,A -85,B 0,C 180,E1 -26510.751,E2 -26510.751} C_VEL
LIN {X 0,Y 98.585,Z 550.19,A -85,B 0,C 180,E1 -26515.228,E2 -26515.228} C_VEL
LIN {X 0,Y 97.714,Z 549.813,A -85,B 0,C 180,E1 -26519.77,E2 -26519.77} C_VEL
LIN {X 0,Y 97.392,Z 547.756,A -85,B 0,C 180,E1 -26528.85,E2 -26528.85} C_VEL
LIN {X 0,Y 98.288,Z 544.922,A -85,B 0,C 180,E1 -26535.507,E2 -26535.507} C_VEL
LIN {X 0,Y 100.014,Z 540.964,A -85,B 0,C 180,E1 -26541.921,E2 -26541.921} C_VEL
LIN {X 0,Y 101.565,Z 537.739,A -85,B 0,C 180,E1 -26546.033,E2 -26546.033} C_VEL
LIN {X 0,Y 104.696,Z 531.751,A -85,B 0,C 180,E1 -26551.873,E2 -26551.873} C_VEL
LIN {X 0,Y 108.759,Z 524.008,A -85,B 0,C 180,E1 -26557.426,E2 -26557.426} C_VEL
LIN {X 0,Y 112.807,Z 516.17,A -85,B 0,C 180,E1 -26561.682,E2 -26561.682} C_VEL
LIN {X 0,Y 116.336,Z 508.808,A -85,B 0,C 180,E1 -26564.853,E2 -26564.853} C_VEL
LIN {X 0,Y 120.383,Z 499.819,A -85,B 0,C 180,E1 -26567.849,E2 -26567.849} C_VEL
LIN {X 0,Y 124.055,Z 490.436,A -85,B 0,C 180,E1 -26570.304,E2 -26570.304} C_VEL
LIN {X 0,Y 127.334,Z 480.657,A -85,B 0,C 180,E1 -26572.3,E2 -26572.3} C_VEL
LIN {X 0,Y 130.272,Z 470.104,A -85,B 0,C 180,E1 -26573.939,E2 -26573.939} C_VEL
LIN {X 0,Y 132.624,Z 458.938,A -85,B 0,C 180,E1 -26575.241,E2 -26575.241} C_VEL
LIN {X 0,Y 134.399,Z 448.449,A -85,B 0,C 180,E1 -26576.046,E2 -26576.046} C_VEL
LIN {X 0,Y 136.307,Z 429.243,A -85,B 0,C 180,E1 -26576.971,E2 -26576.971} C_VEL
LIN {X 0,Y 137.911,Z 409.106,A -85,B 0,C 180,E1 -26577.871,E2 -26577.871} C_VEL
LIN {X 0,Y 134.833,Z 401.303,A -85,B 0,C 180,E1 -26579.775,E2 -26579.775} C_VEL
LIN {X 0,Y 129.926,Z 391.771,A -85,B 0,C 180,E1 -26582.9,E2 -26582.9} C_VEL
LIN {X 0,Y 124.447,Z 382.337,A -85,B 0,C 180,E1 -26586.757,E2 -26586.757} C_VEL
LIN {X 0,Y 119.939,Z 375.448,A -85,B 0,C 180,E1 -26590.38,E2 -26590.38} C_VEL
LIN {X 0,Y 116.42,Z 370.518,A -85,B 0,C 180,E1 -26593.579,E2 -26593.579} C_VEL
LIN {X 0,Y 113.59,Z 366.67,A -85,B 0,C 180,E1 -26596.501,E2 -26596.501} C_VEL
LIN {X 0,Y 111.075,Z 363.746,A -85,B 0,C 180,E1 -26599.356,E2 -26599.356} C_VEL
LIN {X 0,Y 109.947,Z 361.767,A -85,B 0,C 180,E1 -26600.889,E2 -26600.889} C_VEL
LIN {X 0,Y 107.216,Z 359.325,A -85,B 0,C 180,E1 -26604.713,E2 -26604.713} C_VEL
LIN {X 0,Y 105.524,Z 356.337,A -85,B 0,C 180,E1 -26607.804,E2 -26607.804} C_VEL
LIN {X 0,Y 102.276,Z 354.014,A -85,B 0,C 180,E1 -26615.054,E2 -26615.054} C_VEL
LIN {X 0,Y 101.052,Z 351.528,A -85,B 0,C 180,E1 -26620.709,E2 -26620.709} C_VEL
LIN {X 0,Y 101.092,Z 350.677,A -85,B 0,C 180,E1 -26626.731,E2 -26626.731} C_VEL
LIN {X 0,Y 101.337,Z 350.777,A -85,B 0,C 180,E1 -26634.028,E2 -26634.028} C_VEL
LIN {X 0,Y 102.29,Z 352.033,A -85,B 0,C 180,E1 -26639.999,E2 -26639.999} C_VEL
LIN {X 0,Y 103.313,Z 354.333,A -85,B 0,C 180,E1 -26643.411,E2 -26643.411} C_VEL
LIN {X 0,Y 106.364,Z 356.74,A -85,B 0,C 180,E1 -26649.387,E2 -26649.387} C_VEL
LIN {X 0,Y 108.153,Z 360.042,A -85,B 0,C 180,E1 -26652.484,E2 -26652.484} C_VEL
LIN {X 0,Y 110.368,Z 362.143,A -85,B 0,C 180,E1 -26655.464,E2 -26655.464} C_VEL
LIN {X 0,Y 112.41,Z 365.346,A -85,B 0,C 180,E1 -26658.039,E2 -26658.039} C_VEL
LIN {X 0,Y 114.192,Z 367.258,A -85,B 0,C 180,E1 -26659.946,E2 -26659.946} C_VEL
LIN {X 0,Y 116.807,Z 370.941,A -85,B 0,C 180,E1 -26662.6,E2 -26662.6} C_VEL
LIN {X 0,Y 121.169,Z 377.29,A -85,B 0,C 180,E1 -26666.479,E2 -26666.479} C_VEL
LIN {X 0,Y 126.686,Z 386.218,A -85,B 0,C 180,E1 -26670.72,E2 -26670.72} C_VEL
LIN {X 0,Y 130.781,Z 393.835,A -85,B 0,C 180,E1 -26673.538,E2 -26673.538} C_VEL
LIN {X 0,Y 135.231,Z 405.302,A -85,B 0,C 180,E1 -26676.542,E2 -26676.542} C_VEL
LIN {X 0,Y 137.693,Z 412.861,A -85,B 0,C 180,E1 -26678.151,E2 -26678.151} C_VEL
LIN {X 0,Y 134.683,Z 447.793,A -85,B 0,C 180,E1 -26679.745,E2 -26679.745} C_VEL
LIN {X 0,Y 133.244,Z 458.167,A -85,B 0,C 180,E1 -26680.471,E2 -26680.471} C_VEL
LIN {X 0,Y 131.266,Z 468.117,A -85,B 0,C 180,E1 -26681.447,E2 -26681.447} C_VEL
LIN {X 0,Y 128.871,Z 477.23,A -85,B 0,C 180,E1 -26682.589,E2 -26682.589} C_VEL
LIN {X 0,Y 125.641,Z 488.001,A -85,B 0,C 180,E1 -26684.504,E2 -26684.504} C_VEL
LIN {X 0,Y 122.355,Z 496.78,A -85,B 0,C 180,E1 -26686.427,E2 -26686.427} C_VEL
LIN {X 0,Y 118.344,Z 506.403,A -85,B 0,C 180,E1 -26689.213,E2 -26689.213} C_VEL
LIN {X 0,Y 114.63,Z 514.466,A -85,B 0,C 180,E1 -26692.185,E2 -26692.185} C_VEL
LIN {X 0,Y 110.127,Z 523.365,A -85,B 0,C 180,E1 -26696.487,E2 -26696.487} C_VEL
LIN {X 0,Y 106.835,Z 529.736,A -85,B 0,C 180,E1 -26700.437,E2 -26700.437} C_VEL
LIN {X 0,Y 103.812,Z 535.521,A -85,B 0,C 180,E1 -26704.968,E2 -26704.968} C_VEL
LIN {X 0,Y 101.312,Z 540.311,A -85,B 0,C 180,E1 -26709.705,E2 -26709.705} C_VEL
LIN {X 0,Y 99.375,Z 544.888,A -85,B 0,C 180,E1 -26715.668,E2 -26715.668} C_VEL
LIN {X 0,Y 98.243,Z 548.34,A -85,B 0,C 180,E1 -26721.774,E2 -26721.774} C_VEL
LIN {X 0,Y 97.942,Z 551.281,A -85,B 0,C 180,E1 -26730,E2 -26730} C_VEL
LIN {X 0,Y 97.948,Z 552.218,A -85,B 0,C 180,E1 -26734.114,E2 -26734.114} C_VEL
LIN {X 0,Y 98.955,Z 552.759,A -85,B 0,C 180,E1 -26742.302,E2 -26742.302} C_VEL
LIN {X 0,Y 101.625,Z 551.712,A -85,B 0,C 180,E1 -26750.229,E2 -26750.229} C_VEL
LIN {X 0,Y 103.573,Z 550.727,A -85,B 0,C 180,E1 -26754.024,E2 -26754.024} C_VEL
LIN {X 0,Y 109.019,Z 547.308,A -85,B 0,C 180,E1 -26761.046,E2 -26761.046} C_VEL
LIN {X 0,Y 113.961,Z 543.677,A -85,B 0,C 180,E1 -26765.864,E2 -26765.864} C_VEL
LIN {X 0,Y 119.584,Z 538.976,A -85,B 0,C 180,E1 -26770.276,E2 -26770.276} C_VEL
LIN {X 0,Y 125.994,Z 533.044,A -85,B 0,C 180,E1 -26774.207,E2 -26774.207} C_VEL
LIN {X 0,Y 131.775,Z 527.07,A -85,B 0,C 180,E1 -26777.166,E2 -26777.166} C_VEL
LIN {X 0,Y 137.917,Z 519.895,A -85,B 0,C 180,E1 -26779.851,E2 -26779.851} C_VEL
LIN {X 0,Y 144.3,Z 511.245,A -85,B 0,C 180,E1 -26782.32,E2 -26782.32} C_VEL
LIN {X 0,Y 150.333,Z 501.793,A -85,B 0,C 180,E1 -26784.318,E2 -26784.318} C_VEL
LIN {X 0,Y 155.125,Z 492.993,A -85,B 0,C 180,E1 -26785.773,E2 -26785.773} C_VEL
LIN {X 0,Y 159.31,Z 483.951,A -85,B 0,C 180,E1 -26786.949,E2 -26786.949} C_VEL
LIN {X 0,Y 163.589,Z 472.472,A -85,B 0,C 180,E1 -26788.047,E2 -26788.047} C_VEL
LIN {X 0,Y 164.62,Z 469.164,A -85,B 0,C 180,E1 -26788.291,E2 -26788.291} C_VEL
LIN {X 0,Y 166.053,Z 463.658,A -85,B 0,C 180,E1 -26788.861,E2 -26788.861} C_VEL
LIN {X 0,Y 167.041,Z 454.691,A -85,B 0,C 180,E1 -26790.297,E2 -26790.297} C_VEL
LIN {X 0,Y 167.57,Z 445.557,A -85,B 0,C 180,E1 -26791.605,E2 -26791.605} C_VEL
LIN {X 0,Y 168.073,Z 439.791,A -85,B 0,C 180,E1 -26792.001,E2 -26792.001} C_VEL
LIN {X 0,Y 168.384,Z 436.718,A -85,B 0,C 180,E1 -26792.126,E2 -26792.126} C_VEL
LIN {X 0,Y 166.769,Z 431.211,A -85,B 0,C 180,E1 -26794.865,E2 -26794.865} C_VEL
LIN {X 0,Y 165.976,Z 429.27,A -85,B 0,C 180,E1 -26796.281,E2 -26796.281} C_VEL
LIN {X 0,Y 164.81,Z 426.626,A -85,B 0,C 180,E1 -26798.768,E2 -26798.768} C_VEL
LIN {X 0,Y 163.583,Z 423.681,A -85,B 0,C 180,E1 -26802.499,E2 -26802.499} C_VEL
LIN {X 0,Y 162.858,Z 422.529,A -85,B 0,C 180,E1 -26807.54,E2 -26807.54} C_VEL
LIN {X 0,Y 163.052,Z 422.697,A -85,B 0,C 180,E1 -26810.855,E2 -26810.855} C_VEL
LIN {X 0,Y 163.954,Z 423.891,A -85,B 0,C 180,E1 -26814.844,E2 -26814.844} C_VEL
LIN {X 0,Y 165.667,Z 427.978,A -85,B 0,C 180,E1 -26819.267,E2 -26819.267} C_VEL
LIN {X 0,Y 167.596,Z 432.611,A -85,B 0,C 180,E1 -26822.621,E2 -26822.621} C_VEL
LIN {X 0,Y 168.555,Z 435.065,A -85,B 0,C 180,E1 -26824.059,E2 -26824.059} C_VEL
LIN {X 0,Y 166.192,Z 452.09,A -85,B 0,C 180,E1 -26824.655,E2 -26824.655} C_VEL
LIN {X 0,Y 162.88,Z 465.371,A -85,B 0,C 180,E1 -26825.409,E2 -26825.409} C_VEL
LIN {X 0,Y 159.105,Z 476.571,A -85,B 0,C 180,E1 -26826.348,E2 -26826.348} C_VEL
LIN {X 0,Y 154.965,Z 486.325,A -85,B 0,C 180,E1 -26827.415,E2 -26827.415} C_VEL
LIN {X 0,Y 150.519,Z 495.118,A -85,B 0,C 180,E1 -26828.668,E2 -26828.668} C_VEL
LIN {X 0,Y 144.707,Z 504.697,A -85,B 0,C 180,E1 -26830.428,E2 -26830.428} C_VEL
LIN {X 0,Y 138.398,Z 513.519,A -85,B 0,C 180,E1 -26832.569,E2 -26832.569} C_VEL
LIN {X 0,Y 132.665,Z 520.547,A -85,B 0,C 180,E1 -26834.805,E2 -26834.805} C_VEL
LIN {X 0,Y 125.569,Z 528.001,A -85,B 0,C 180,E1 -26837.923,E2 -26837.923} C_VEL
LIN {X 0,Y 118.909,Z 534.111,A -85,B 0,C 180,E1 -26841.427,E2 -26841.427} C_VEL
LIN {X 0,Y 113.185,Z 538.791,A -85,B 0,C 180,E1 -26845.067,E2 -26845.067} C_VEL
LIN {X 0,Y 108.247,Z 542.405,A -85,B 0,C 180,E1 -26848.778,E2 -26848.778} C_VEL
LIN {X 0,Y 102.345,Z 546.13,A -85,B 0,C 180,E1 -26854.51,E2 -26854.51} C_VEL
LIN {X 0,Y 97.876,Z 548.485,A -85,B 0,C 180,E1 -26860.261,E2 -26860.261} C_VEL
LIN {X 0,Y 93.467,Z 550.042,A -85,B 0,C 180,E1 -26868.759,E2 -26868.759} C_VEL
LIN {X 0,Y 92.161,Z 550.295,A -85,B 0,C 180,E1 -26872.407,E2 -26872.407} C_VEL
LIN {X 0,Y 90.796,Z 549.937,A -85,B 0,C 180,E1 -26878.371,E2 -26878.371} C_VEL
LIN {X 0,Y 90.212,Z 548.296,A -85,B 0,C 180,E1 -26887.075,E2 -26887.075} C_VEL
LIN {X 0,Y 90.903,Z 545.683,A -85,B 0,C 180,E1 -26894.301,E2 -26894.301} C_VEL
LIN {X 0,Y 92.596,Z 541.95,A -85,B 0,C 180,E1 -26901.269,E2 -26901.269} C_VEL
LIN {X 0,Y 95.594,Z 536.007,A -85,B 0,C 180,E1 -26908.947,E2 -26908.947} C_VEL
LIN {X 0,Y 98.662,Z 530.528,A -85,B 0,C 180,E1 -26914.23,E2 -26914.23} C_VEL
LIN {X 0,Y 102.215,Z 524.27,A -85,B 0,C 180,E1 -26918.9,E2 -26918.9} C_VEL
LIN {X 0,Y 106.494,Z 516.462,A -85,B 0,C 180,E1 -26923.355,E2 -26923.355} C_VEL
LIN {X 0,Y 110.364,Z 508.772,A -85,B 0,C 180,E1 -26926.794,E2 -26926.794} C_VEL
LIN {X 0,Y 114.438,Z 500.204,A -85,B 0,C 180,E1 -26929.742,E2 -26929.742} C_VEL
LIN {X 0,Y 118.289,Z 490.878,A -85,B 0,C 180,E1 -26932.257,E2 -26932.257} C_VEL
LIN {X 0,Y 121.794,Z 480.977,A -85,B 0,C 180,E1 -26934.322,E2 -26934.322} C_VEL
LIN {X 0,Y 124.804,Z 470.668,A -85,B 0,C 180,E1 -26935.967,E2 -26935.967} C_VEL
LIN {X 0,Y 127.289,Z 459.605,A -85,B 0,C 180,E1 -26937.285,E2 -26937.285} C_VEL
LIN {X 0,Y 129.252,Z 448.263,A -85,B 0,C 180,E1 -26938.169,E2 -26938.169} C_VEL
LIN {X 0,Y 131.163,Z 429.705,A -85,B 0,C 180,E1 -26939.071,E2 -26939.071} C_VEL
LIN {X 0,Y 132.688,Z 411.099,A -85,B 0,C 180,E1 -26939.925,E2 -26939.925} C_VEL
LIN {X 0,Y 130.287,Z 404.976,A -85,B 0,C 180,E1 -26941.56,E2 -26941.56} C_VEL
LIN {X 0,Y 124.83,Z 394.277,A -85,B 0,C 180,E1 -26945.363,E2 -26945.363} C_VEL
LIN {X 0,Y 119.513,Z 385.046,A -85,B 0,C 180,E1 -26949.614,E2 -26949.614} C_VEL
LIN {X 0,Y 116.449,Z 380.466,A -85,B 0,C 180,E1 -26952.336,E2 -26952.336} C_VEL
LIN {X 0,Y 113.464,Z 376.113,A -85,B 0,C 180,E1 -26955.321,E2 -26955.321} C_VEL
LIN {X 0,Y 111.255,Z 372.927,A -85,B 0,C 180,E1 -26957.807,E2 -26957.807} C_VEL
LIN {X 0,Y 108.713,Z 369.665,A -85,B 0,C 180,E1 -26960.987,E2 -26960.987} C_VEL
LIN {X 0,Y 107.901,Z 368.284,A -85,B 0,C 180,E1 -26962.175,E2 -26962.175} C_VEL
LIN {X 0,Y 105.167,Z 365.407,A -85,B 0,C 180,E1 -26966.397,E2 -26966.397} C_VEL
LIN {X 0,Y 104.01,Z 363.097,A -85,B 0,C 180,E1 -26968.75,E2 -26968.75} C_VEL
LIN {X 0,Y 101.144,Z 360.961,A -85,B 0,C 180,E1 -26975.576,E2 -26975.576} C_VEL
LIN {X 0,Y 99.792,Z 358.252,A -85,B 0,C 180,E1 -26982.053,E2 -26982.053} C_VEL
LIN {X 0,Y 99.442,Z 357.525,A -85,B 0,C 180,E1 -26987.758,E2 -26987.758} C_VEL
LIN {X 0,Y 99.893,Z 357.711,A -85,B 0,C 180,E1 -26993.941,E2 -26993.941} C_VEL
LIN {X 0,Y 101.061,Z 359.081,A -85,B 0,C 180,E1 -26999.252,E2 -26999.252} C_VEL
LIN {X 0,Y 102.155,Z 361.339,A -85,B 0,C 180,E1 -27002.957,E2 -27002.957} C_VEL
LIN {X 0,Y 104.595,Z 363.299,A -85,B 0,C 180,E1 -27008.086,E2 -27008.086} C_VEL
LIN {X 0,Y 106.402,Z 366.611,A -85,B 0,C 180,E1 -27011.428,E2 -27011.428} C_VEL
LIN {X 0,Y 108.264,Z 368.533,A -85,B 0,C 180,E1 -27014.126,E2 -27014.126} C_VEL
LIN {X 0,Y 110.602,Z 372.073,A -85,B 0,C 180,E1 -27017.244,E2 -27017.244} C_VEL
LIN {X 0,Y 111.905,Z 373.717,A -85,B 0,C 180,E1 -27018.749,E2 -27018.749} C_VEL
LIN {X 0,Y 115.187,Z 378.507,A -85,B 0,C 180,E1 -27022.259,E2 -27022.259} C_VEL
LIN {X 0,Y 119.04,Z 384.347,A -85,B 0,C 180,E1 -27025.811,E2 -27025.811} C_VEL
LIN {X 0,Y 124.562,Z 394.002,A -85,B 0,C 180,E1 -27030.282,E2 -27030.282} C_VEL
LIN {X 0,Y 127.038,Z 399.101,A -85,B 0,C 180,E1 -27032.107,E2 -27032.107} C_VEL
LIN {X 0,Y 131.099,Z 410.238,A -85,B 0,C 180,E1 -27035.101,E2 -27035.101} C_VEL
LIN {X 0,Y 132.532,Z 414.844,A -85,B 0,C 180,E1 -27036.136,E2 -27036.136} C_VEL
LIN {X 0,Y 129.486,Z 448.007,A -85,B 0,C 180,E1 -27037.655,E2 -27037.655} C_VEL
LIN {X 0,Y 128.069,Z 457.818,A -85,B 0,C 180,E1 -27038.345,E2 -27038.345} C_VEL
LIN {X 0,Y 126.026,Z 467.711,A -85,B 0,C 180,E1 -27039.307,E2 -27039.307} C_VEL
LIN {X 0,Y 122.929,Z 478.754,A -85,B 0,C 180,E1 -27040.753,E2 -27040.753} C_VEL
LIN {X 0,Y 119.551,Z 489.205,A -85,B 0,C 180,E1 -27042.706,E2 -27042.706} C_VEL
LIN {X 0,Y 116.216,Z 497.776,A -85,B 0,C 180,E1 -27044.718,E2 -27044.718} C_VEL
LIN {X 0,Y 111.967,Z 507.199,A -85,B 0,C 180,E1 -27047.564,E2 -27047.564} C_VEL
LIN {X 0,Y 108.125,Z 515.122,A -85,B 0,C 180,E1 -27050.673,E2 -27050.673} C_VEL
LIN {X 0,Y 104.289,Z 522.261,A -85,B 0,C 180,E1 -27054.179,E2 -27054.179} C_VEL
LIN {X 0,Y 100.694,Z 528.971,A -85,B 0,C 180,E1 -27058.434,E2 -27058.434} C_VEL
LIN {X 0,Y 96.795,Z 535.846,A -85,B 0,C 180,E1 -27064.173,E2 -27064.173} C_VEL
LIN {X 0,Y 93.829,Z 541.341,A -85,B 0,C 180,E1 -27070.302,E2 -27070.302} C_VEL
LIN {X 0,Y 91.957,Z 545.636,A -85,B 0,C 180,E1 -27076.745,E2 -27076.745} C_VEL
LIN {X 0,Y 91.215,Z 547.953,A -85,B 0,C 180,E1 -27081.135,E2 -27081.135} C_VEL
LIN {X 0,Y 90.841,Z 551.046,A -85,B 0,C 180,E1 -27090,E2 -27090} C_VEL
LIN {X 0,Y 90.879,Z 551.983,A -85,B 0,C 180,E1 -27094.435,E2 -27094.435} C_VEL
LIN {X 0,Y 92.029,Z 552.696,A -85,B 0,C 180,E1 -27103.244,E2 -27103.244} C_VEL
LIN {X 0,Y 94.959,Z 551.756,A -85,B 0,C 180,E1 -27111.719,E2 -27111.719} C_VEL
LIN {X 0,Y 97.111,Z 550.785,A -85,B 0,C 180,E1 -27115.736,E2 -27115.736} C_VEL
LIN {X 0,Y 103.014,Z 547.559,A -85,B 0,C 180,E1 -27123.078,E2 -27123.078} C_VEL
LIN {X 0,Y 108.283,Z 544.037,A -85,B 0,C 180,E1 -27128.067,E2 -27128.067} C_VEL
LIN {X 0,Y 114.279,Z 539.451,A -85,B 0,C 180,E1 -27132.569,E2 -27132.569} C_VEL
LIN {X 0,Y 121.044,Z 533.665,A -85,B 0,C 180,E1 -27136.533,E2 -27136.533} C_VEL
LIN {X 0,Y 128.325,Z 526.472,A -85,B 0,C 180,E1 -27140.061,E2 -27140.061} C_VEL
LIN {X 0,Y 134.766,Z 519.229,A -85,B 0,C 180,E1 -27142.681,E2 -27142.681} C_VEL
LIN {X 0,Y 141.501,Z 510.459,A -85,B 0,C 180,E1 -27145.036,E2 -27145.036} C_VEL
LIN {X 0,Y 147.064,Z 502.073,A -85,B 0,C 180,E1 -27146.751,E2 -27146.751} C_VEL
LIN {X 0,Y 152.729,Z 491.895,A -85,B 0,C 180,E1 -27148.353,E2 -27148.353} C_VEL
LIN {X 0,Y 157.063,Z 482.607,A -85,B 0,C 180,E1 -27149.47,E2 -27149.47} C_VEL
LIN {X 0,Y 161.119,Z 471.929,A -85,B 0,C 180,E1 -27150.42,E2 -27150.42} C_VEL
LIN {X 0,Y 164.296,Z 461.229,A -85,B 0,C 180,E1 -27151.095,E2 -27151.095} C_VEL
LIN {X 0,Y 166.653,Z 449.9,A -85,B 0,C 180,E1 -27151.649,E2 -27151.649} C_VEL
LIN {X 0,Y 168.073,Z 439.791,A -85,B 0,C 180,E1 -27152.001,E2 -27152.001} C_VEL
LIN {X 0,Y 168.051,Z 437.747,A -85,B 0,C 180,E1 -27152.327,E2 -27152.327} C_VEL
LIN {X 0,Y 167.546,Z 436.001,A -85,B 0,C 180,E1 -27153.147,E2 -27153.147} C_VEL
LIN {X 0,Y 166.471,Z 434.857,A -85,B 0,C 180,E1 -27154.609,E2 -27154.609} C_VEL
LIN {X 0,Y 164.009,Z 434.133,A -85,B 0,C 180,E1 -27158.37,E2 -27158.37} C_VEL
LIN {X 0,Y 163.768,Z 433.78,A -85,B 0,C 180,E1 -27158.904,E2 -27158.904} C_VEL
LIN {X 0,Y 162.539,Z 430.638,A -85,B 0,C 180,E1 -27162.864,E2 -27162.864} C_VEL
LIN {X 0,Y 161.92,Z 429.585,A -85,B 0,C 180,E1 -27167.467,E2 -27167.467} C_VEL
LIN {X 0,Y 162.104,Z 429.727,A -85,B 0,C 180,E1 -27170.801,E2 -27170.801} C_VEL
LIN {X 0,Y 162.835,Z 430.769,A -85,B 0,C 180,E1 -27174.341,E2 -27174.341} C_VEL
LIN {X 0,Y 164.307,Z 434.625,A -85,B 0,C 180,E1 -27178.521,E2 -27178.521} C_VEL
LIN {X 0,Y 166.04,Z 439.282,A -85,B 0,C 180,E1 -27181.869,E2 -27181.869} C_VEL
LIN {X 0,Y 163.544,Z 454.434,A -85,B 0,C 180,E1 -27182.411,E2 -27182.411} C_VEL
LIN {X 0,Y 160.552,Z 465.827,A -85,B 0,C 180,E1 -27183.042,E2 -27183.042} C_VEL
LIN {X 0,Y 156.739,Z 476.744,A -85,B 0,C 180,E1 -27183.92,E2 -27183.92} C_VEL
LIN {X 0,Y 152.5,Z 486.403,A -85,B 0,C 180,E1 -27184.926,E2 -27184.926} C_VEL
LIN {X 0,Y 147.571,Z 495.708,A -85,B 0,C 180,E1 -27186.194,E2 -27186.194} C_VEL
LIN {X 0,Y 141.868,Z 504.745,A -85,B 0,C 180,E1 -27187.787,E2 -27187.787} C_VEL
LIN {X 0,Y 135.505,Z 513.34,A -85,B 0,C 180,E1 -27189.79,E2 -27189.79} C_VEL
LIN {X 0,Y 129.333,Z 520.594,A -85,B 0,C 180,E1 -27192.006,E2 -27192.006} C_VEL
LIN {X 0,Y 121.888,Z 528.052,A -85,B 0,C 180,E1 -27195.03,E2 -27195.03} C_VEL
LIN {X 0,Y 116.696,Z 532.753,A -85,B 0,C 180,E1 -27197.526,E2 -27197.526} C_VEL
LIN {X 0,Y 109.559,Z 538.305,A -85,B 0,C 180,E1 -27201.543,E2 -27201.543} C_VEL
LIN {X 0,Y 102.281,Z 543.117,A -85,B 0,C 180,E1 -27206.714,E2 -27206.714} C_VEL
LIN {X 0,Y 97.982,Z 545.661,A -85,B 0,C 180,E1 -27210.602,E2 -27210.602} C_VEL
LIN {X 0,Y 91.963,Z 548.588,A -85,B 0,C 180,E1 -27217.69,E2 -27217.69} C_VEL
LIN {X 0,Y 88.119,Z 549.964,A -85,B 0,C 180,E1 -27224.127,E2 -27224.127} C_VEL
LIN {X 0,Y 86.002,Z 550.308,A -85,B 0,C 180,E1 -27229.175,E2 -27229.175} C_VEL
LIN {X 0,Y 83.487,Z 549.769,A -85,B 0,C 180,E1 -27239.664,E2 -27239.664} C_VEL
LIN {X 0,Y 83.157,Z 547.803,A -85,B 0,C 180,E1 -27248.385,E2 -27248.385} C_VEL
LIN {X 0,Y 83.988,Z 545.256,A -85,B 0,C 180,E1 -27255.462,E2 -27255.462} C_VEL
LIN {X 0,Y 85.987,Z 541.115,A -85,B 0,C 180,E1 -27263.279,E2 -27263.279} C_VEL
LIN {X 0,Y 88.684,Z 536.208,A -85,B 0,C 180,E1 -27270,E2 -27270} C_VEL
LIN {X 0,Y 91.765,Z 531.088,A -85,B 0,C 180,E1 -27275.35,E2 -27275.35} C_VEL
LIN {X 0,Y 95.74,Z 524.522,A -85,B 0,C 180,E1 -27280.575,E2 -27280.575} C_VEL
LIN {X 0,Y 100.26,Z 516.749,A -85,B 0,C 180,E1 -27285.241,E2 -27285.241} C_VEL
LIN {X 0,Y 104.652,Z 508.511,A -85,B 0,C 180,E1 -27289.03,E2 -27289.03} C_VEL
LIN {X 0,Y 108.653,Z 500.571,A -85,B 0,C 180,E1 -27291.835,E2 -27291.835} C_VEL
LIN {X 0,Y 112.68,Z 491.312,A -85,B 0,C 180,E1 -27294.407,E2 -27294.407} C_VEL
LIN {X 0,Y 116.272,Z 481.696,A -85,B 0,C 180,E1 -27296.474,E2 -27296.474} C_VEL
LIN {X 0,Y 119.714,Z 470.405,A -85,B 0,C 180,E1 -27298.284,E2 -27298.284} C_VEL
LIN {X 0,Y 122.326,Z 459.136,A -85,B 0,C 180,E1 -27299.617,E2 -27299.617} C_VEL
LIN {X 0,Y 124.236,Z 448.478,A -85,B 0,C 180,E1 -27300.446,E2 -27300.446} C_VEL
LIN {X 0,Y 126.171,Z 430.635,A -85,B 0,C 180,E1 -27301.317,E2 -27301.317} C_VEL
LIN {X 0,Y 127.725,Z 413.268,A -85,B 0,C 180,E1 -27302.092,E2 -27302.092} C_VEL
LIN {X 0,Y 124.606,Z 406.039,A -85,B 0,C 180,E1 -27304.362,E2 -27304.362} C_VEL
LIN {X 0,Y 119.236,Z 395.609,A -85,B 0,C 180,E1 -27308.639,E2 -27308.639} C_VEL
LIN {X 0,Y 114.519,Z 387.439,A -85,B 0,C 180,E1 -27312.975,E2 -27312.975} C_VEL
LIN {X 0,Y 110.48,Z 381.422,A -85,B 0,C 180,E1 -27317.328,E2 -27317.328} C_VEL
LIN {X 0,Y 108.904,Z 379.112,A -85,B 0,C 180,E1 -27319.259,E2 -27319.259} C_VEL
LIN {X 0,Y 106.228,Z 375.196,A -85,B 0,C 180,E1 -27322.999,E2 -27322.999} C_VEL
LIN {X 0,Y 103.14,Z 371.38,A -85,B 0,C 180,E1 -27328.271,E2 -27328.271} C_VEL
LIN {X 0,Y 102.437,Z 369.893,A -85,B 0,C 180,E1 -27329.878,E2 -27329.878} C_VEL
LIN {X 0,Y 99.649,Z 367.353,A -85,B 0,C 180,E1 -27337.478,E2 -27337.478} C_VEL
LIN {X 0,Y 98.742,Z 365.147,A -85,B 0,C 180,E1 -27342.926,E2 -27342.926} C_VEL
LIN {X 0,Y 98.503,Z 364.581,A -85,B 0,C 180,E1 -27347.64,E2 -27347.64} C_VEL
LIN {X 0,Y 98.949,Z 364.772,A -85,B 0,C 180,E1 -27353.923,E2 -27353.923} C_VEL
LIN {X 0,Y 99.773,Z 365.781,A -85,B 0,C 180,E1 -27358.044,E2 -27358.044} C_VEL
LIN {X 0,Y 101.052,Z 368.342,A -85,B 0,C 180,E1 -27362.615,E2 -27362.615} C_VEL
LIN {X 0,Y 102.983,Z 370.115,A -85,B 0,C 180,E1 -27366.981,E2 -27366.981} C_VEL
LIN {X 0,Y 104.951,Z 373.544,A -85,B 0,C 180,E1 -27370.794,E2 -27370.794} C_VEL
LIN {X 0,Y 106.337,Z 375.162,A -85,B 0,C 180,E1 -27372.956,E2 -27372.956} C_VEL
LIN {X 0,Y 108.922,Z 378.932,A -85,B 0,C 180,E1 -27376.557,E2 -27376.557} C_VEL
LIN {X 0,Y 112.575,Z 384.508,A -85,B 0,C 180,E1 -27380.857,E2 -27380.857} C_VEL
LIN {X 0,Y 116.153,Z 390.272,A -85,B 0,C 180,E1 -27384.434,E2 -27384.434} C_VEL
LIN {X 0,Y 121.058,Z 399.236,A -85,B 0,C 180,E1 -27388.734,E2 -27388.734} C_VEL
LIN {X 0,Y 123.147,Z 403.785,A -85,B 0,C 180,E1 -27390.43,E2 -27390.43} C_VEL
LIN {X 0,Y 126.959,Z 414.886,A -85,B 0,C 180,E1 -27393.494,E2 -27393.494} C_VEL
LIN {X 0,Y 127.503,Z 416.691,A -85,B 0,C 180,E1 -27393.929,E2 -27393.929} C_VEL
LIN {X 0,Y 124.478,Z 448.133,A -85,B 0,C 180,E1 -27395.384,E2 -27395.384} C_VEL
LIN {X 0,Y 122.962,Z 458.069,A -85,B 0,C 180,E1 -27396.094,E2 -27396.094} C_VEL
LIN {X 0,Y 120.681,Z 468.519,A -85,B 0,C 180,E1 -27397.145,E2 -27397.145} C_VEL
LIN {X 0,Y 117.766,Z 478.422,A -85,B 0,C 180,E1 -27398.438,E2 -27398.438} C_VEL
LIN {X 0,Y 114.227,Z 488.919,A -85,B 0,C 180,E1 -27400.412,E2 -27400.412} C_VEL
LIN {X 0,Y 110.729,Z 497.523,A -85,B 0,C 180,E1 -27402.452,E2 -27402.452} C_VEL
LIN {X 0,Y 106.265,Z 506.973,A -85,B 0,C 180,E1 -27405.355,E2 -27405.355} C_VEL
LIN {X 0,Y 101.728,Z 515.782,A -85,B 0,C 180,E1 -27408.98,E2 -27408.98} C_VEL
LIN {X 0,Y 98.062,Z 522.17,A -85,B 0,C 180,E1 -27412.249,E2 -27412.249} C_VEL
LIN {X 0,Y 93.888,Z 529.391,A -85,B 0,C 180,E1 -27417.132,E2 -27417.132} C_VEL
LIN {X 0,Y 90.446,Z 535.204,A -85,B 0,C 180,E1 -27422.21,E2 -27422.21} C_VEL
LIN {X 0,Y 87.126,Z 540.804,A -85,B 0,C 180,E1 -27428.716,E2 -27428.716} C_VEL
LIN {X 0,Y 85.037,Z 545.204,A -85,B 0,C 180,E1 -27435.644,E2 -27435.644} C_VEL
LIN {X 0,Y 84.195,Z 547.523,A -85,B 0,C 180,E1 -27440.389,E2 -27440.389} C_VEL
LIN {X 0,Y 83.763,Z 550.805,A -85,B 0,C 180,E1 -27450,E2 -27450} C_VEL
LIN {X 0,Y 83.797,Z 551.739,A -85,B 0,C 180,E1 -27454.811,E2 -27454.811} C_VEL
LIN {X 0,Y 85.109,Z 552.594,A -85,B 0,C 180,E1 -27464.343,E2 -27464.343} C_VEL
LIN {X 0,Y 88.368,Z 551.803,A -85,B 0,C 180,E1 -27473.431,E2 -27473.431} C_VEL
LIN {X 0,Y 90.753,Z 550.831,A -85,B 0,C 180,E1 -27477.687,E2 -27477.687} C_VEL
LIN {X 0,Y 97.14,Z 547.793,A -85,B 0,C 180,E1 -27485.365,E2 -27485.365} C_VEL
LIN {X 0,Y 102.788,Z 544.371,A -85,B 0,C 180,E1 -27490.507,E2 -27490.507} C_VEL
LIN {X 0,Y 109.17,Z 539.915,A -85,B 0,C 180,E1 -27495.084,E2 -27495.084} C_VEL
LIN {X 0,Y 117.556,Z 533.174,A -85,B 0,C 180,E1 -27499.663,E2 -27499.663} C_VEL
LIN {X 0,Y 125.241,Z 525.901,A -85,B 0,C 180,E1 -27503.097,E2 -27503.097} C_VEL
LIN {X 0,Y 131.98,Z 518.566,A -85,B 0,C 180,E1 -27505.627,E2 -27505.627} C_VEL
LIN {X 0,Y 138.317,Z 510.676,A -85,B 0,C 180,E1 -27507.642,E2 -27507.642} C_VEL
LIN {X 0,Y 144.077,Z 502.375,A -85,B 0,C 180,E1 -27509.287,E2 -27509.287} C_VEL
LIN {X 0,Y 149.924,Z 492.322,A -85,B 0,C 180,E1 -27510.819,E2 -27510.819} C_VEL
LIN {X 0,Y 154.389,Z 483.195,A -85,B 0,C 180,E1 -27511.881,E2 -27511.881} C_VEL
LIN {X 0,Y 158.676,Z 472.397,A -85,B 0,C 180,E1 -27512.801,E2 -27512.801} C_VEL
LIN {X 0,Y 162.157,Z 461.01,A -85,B 0,C 180,E1 -27513.483,E2 -27513.483} C_VEL
LIN {X 0,Y 164.568,Z 449.795,A -85,B 0,C 180,E1 -27513.992,E2 -27513.992} C_VEL
LIN {X 0,Y 165.91,Z 440.313,A -85,B 0,C 180,E1 -27514.368,E2 -27514.368} C_VEL
LIN {X 0,Y 164.702,Z 436.177,A -85,B 0,C 180,E1 -27516.753,E2 -27516.753} C_VEL
LIN {X 0,Y 163.768,Z 433.78,A -85,B 0,C 180,E1 -27518.904,E2 -27518.904} C_VEL
LIN {X 0,Y 162.941,Z 432.911,A -85,B 0,C 180,E1 -27520.934,E2 -27520.934} C_VEL
LIN {X 0,Y 162.183,Z 433.15,A -85,B 0,C 180,E1 -27523.012,E2 -27523.012} C_VEL
LIN {X 0,Y 161.088,Z 436.601,A -85,B 0,C 180,E1 -27530.066,E2 -27530.066} C_VEL
LIN {X 0,Y 161.716,Z 437.661,A -85,B 0,C 180,E1 -27533.785,E2 -27533.785} C_VEL
LIN {X 0,Y 162.932,Z 441.143,A -85,B 0,C 180,E1 -27537.651,E2 -27537.651} C_VEL
LIN {X 0,Y 163.639,Z 443.635,A -85,B 0,C 180,E1 -27539.583,E2 -27539.583} C_VEL
LIN {X 0,Y 161.534,Z 455.179,A -85,B 0,C 180,E1 -27540.03,E2 -27540.03} C_VEL
LIN {X 0,Y 158.566,Z 466.106,A -85,B 0,C 180,E1 -27540.599,E2 -27540.599} C_VEL
LIN {X 0,Y 154.663,Z 476.941,A -85,B 0,C 180,E1 -27541.412,E2 -27541.412} C_VEL
LIN {X 0,Y 150.41,Z 486.386,A -85,B 0,C 180,E1 -27542.337,E2 -27542.337} C_VEL
LIN {X 0,Y 145.232,Z 495.874,A -85,B 0,C 180,E1 -27543.56,E2 -27543.56} C_VEL
LIN {X 0,Y 139.629,Z 504.504,A -85,B 0,C 180,E1 -27544.975,E2 -27544.975} C_VEL
LIN {X 0,Y 132.752,Z 513.466,A -85,B 0,C 180,E1 -27546.959,E2 -27546.959} C_VEL
LIN {X 0,Y 125.805,Z 521.199,A -85,B 0,C 180,E1 -27549.247,E2 -27549.247} C_VEL
LIN {X 0,Y 118.54,Z 528.123,A -85,B 0,C 180,E1 -27551.973,E2 -27551.973} C_VEL
LIN {X 0,Y 111.36,Z 534.065,A -85,B 0,C 180,E1 -27555.212,E2 -27555.212} C_VEL
LIN {X 0,Y 104.145,Z 539.213,A -85,B 0,C 180,E1 -27559.134,E2 -27559.134} C_VEL
LIN {X 0,Y 98.936,Z 542.533,A -85,B 0,C 180,E1 -27562.563,E2 -27562.563} C_VEL
LIN {X 0,Y 93.766,Z 545.316,A -85,B 0,C 180,E1 -27566.727,E2 -27566.727} C_VEL
LIN {X 0,Y 85.979,Z 548.788,A -85,B 0,C 180,E1 -27575.175,E2 -27575.175} C_VEL
LIN {X 0,Y 82.724,Z 549.829,A -85,B 0,C 180,E1 -27580.128,E2 -27580.128} C_VEL
LIN {X 0,Y 78.123,Z 550.434,A -85,B 0,C 180,E1 -27590.971,E2 -27590.971} C_VEL
LIN {X 0,Y 76.787,Z 550.055,A -85,B 0,C 180,E1 -27596.692,E2 -27596.692} C_VEL
LIN {X 0,Y 76.055,Z 547.746,A -85,B 0,C 180,E1 -27608.308,E2 -27608.308} C_VEL
LIN {X 0,Y 77.098,Z 544.778,A -85,B 0,C 180,E1 -27616.827,E2 -27616.827} C_VEL
LIN {X 0,Y 78.704,Z 541.754,A -85,B 0,C 180,E1 -27623.171,E2 -27623.171} C_VEL
LIN {X 0,Y 81.829,Z 536.373,A -85,B 0,C 180,E1 -27631.231,E2 -27631.231} C_VEL
LIN {X 0,Y 85.818,Z 530.139,A -85,B 0,C 180,E1 -27637.984,E2 -27637.984} C_VEL
LIN {X 0,Y 89.347,Z 524.719,A -85,B 0,C 180,E1 -27642.493,E2 -27642.493} C_VEL
LIN {X 0,Y 94.153,Z 516.963,A -85,B 0,C 180,E1 -27647.373,E2 -27647.373} C_VEL
LIN {X 0,Y 98.911,Z 508.571,A -85,B 0,C 180,E1 -27651.356,E2 -27651.356} C_VEL
LIN {X 0,Y 103.596,Z 499.556,A -85,B 0,C 180,E1 -27654.553,E2 -27654.553} C_VEL
LIN {X 0,Y 107.869,Z 490.05,A -85,B 0,C 180,E1 -27657.134,E2 -27657.134} C_VEL
LIN {X 0,Y 111.651,Z 480.109,A -85,B 0,C 180,E1 -27659.199,E2 -27659.199} C_VEL
LIN {X 0,Y 114.409,Z 471.567,A -85,B 0,C 180,E1 -27660.585,E2 -27660.585} C_VEL
LIN {X 0,Y 117.349,Z 459.558,A -85,B 0,C 180,E1 -27662.03,E2 -27662.03} C_VEL
LIN {X 0,Y 119.373,Z 448.784,A -85,B 0,C 180,E1 -27662.871,E2 -27662.871} C_VEL
LIN {X 0,Y 121.473,Z 430.235,A -85,B 0,C 180,E1 -27663.766,E2 -27663.766} C_VEL
LIN {X 0,Y 122.788,Z 415.335,A -85,B 0,C 180,E1 -27664.473,E2 -27664.473} C_VEL
LIN {X 0,Y 118.713,Z 406.398,A -85,B 0,C 180,E1 -27667.817,E2 -27667.817} C_VEL
LIN {X 0,Y 114.551,Z 398.242,A -85,B 0,C 180,E1 -27671.628,E2 -27671.628} C_VEL
LIN {X 0,Y 111.158,Z 392.406,A -85,B 0,C 180,E1 -27675.14,E2 -27675.14} C_VEL
LIN {X 0,Y 108.15,Z 387.539,A -85,B 0,C 180,E1 -27678.739,E2 -27678.739} C_VEL
LIN {X 0,Y 106.47,Z 385.064,A -85,B 0,C 180,E1 -27680.964,E2 -27680.964} C_VEL
LIN {X 0,Y 104.015,Z 381.233,A -85,B 0,C 180,E1 -27684.799,E2 -27684.799} C_VEL
LIN {X 0,Y 101.436,Z 377.772,A -85,B 0,C 180,E1 -27689.716,E2 -27689.716} C_VEL
LIN {X 0,Y 100.992,Z 376.718,A -85,B 0,C 180,E1 -27690.847,E2 -27690.847} C_VEL
LIN {X 0,Y 98.406,Z 374.037,A -85,B 0,C 180,E1 -27698.686,E2 -27698.686} C_VEL
LIN {X 0,Y 97.761,Z 372.155,A -85,B 0,C 180,E1 -27703.287,E2 -27703.287} C_VEL
LIN {X 0,Y 97.566,Z 371.621,A -85,B 0,C 180,E1 -27707.519,E2 -27707.519} C_VEL
LIN {X 0,Y 97.998,Z 371.833,A -85,B 0,C 180,E1 -27713.864,E2 -27713.864} C_VEL
LIN {X 0,Y 98.584,Z 372.655,A -85,B 0,C 180,E1 -27717.1,E2 -27717.1} C_VEL
LIN {X 0,Y 99.939,Z 375.393,A -85,B 0,C 180,E1 -27722.266,E2 -27722.266} C_VEL
LIN {X 0,Y 101.417,Z 376.876,A -85,B 0,C 180,E1 -27725.841,E2 -27725.841} C_VEL
LIN {X 0,Y 103.483,Z 380.405,A -85,B 0,C 180,E1 -27730.083,E2 -27730.083} C_VEL
LIN {X 0,Y 104.508,Z 381.842,A -85,B 0,C 180,E1 -27731.831,E2 -27731.831} C_VEL
LIN {X 0,Y 107.527,Z 386.533,A -85,B 0,C 180,E1 -27736.27,E2 -27736.27} C_VEL
LIN {X 0,Y 110.361,Z 391.039,A -85,B 0,C 180,E1 -27739.773,E2 -27739.773} C_VEL
LIN {X 0,Y 113.602,Z 396.687,A -85,B 0,C 180,E1 -27743.276,E2 -27743.276} C_VEL
LIN {X 0,Y 117.756,Z 404.643,A -85,B 0,C 180,E1 -27747.189,E2 -27747.189} C_VEL
LIN {X 0,Y 119.609,Z 409.239,A -85,B 0,C 180,E1 -27748.875,E2 -27748.875} C_VEL
LIN {X 0,Y 122.628,Z 418.614,A -85,B 0,C 180,E1 -27751.574,E2 -27751.574} C_VEL
LIN {X 0,Y 119.601,Z 448.592,A -85,B 0,C 180,E1 -27752.976,E2 -27752.976} C_VEL
LIN {X 0,Y 118.004,Z 458.466,A -85,B 0,C 180,E1 -27753.701,E2 -27753.701} C_VEL
LIN {X 0,Y 115.842,Z 467.925,A -85,B 0,C 180,E1 -27754.631,E2 -27754.631} C_VEL
LIN {X 0,Y 112.817,Z 477.933,A -85,B 0,C 180,E1 -27755.919,E2 -27755.919} C_VEL
LIN {X 0,Y 109.104,Z 488.504,A -85,B 0,C 180,E1 -27757.899,E2 -27757.899} C_VEL
LIN {X 0,Y 104.796,Z 498.386,A -85,B 0,C 180,E1 -27760.283,E2 -27760.283} C_VEL
LIN {X 0,Y 100.738,Z 506.652,A -85,B 0,C 180,E1 -27762.9,E2 -27762.9} C_VEL
LIN {X 0,Y 96.42,Z 514.629,A -85,B 0,C 180,E1 -27766.175,E2 -27766.175} C_VEL
LIN {X 0,Y 91.273,Z 523.171,A -85,B 0,C 180,E1 -27770.845,E2 -27770.845} C_VEL
LIN {X 0,Y 87.145,Z 529.754,A -85,B 0,C 180,E1 -27775.63,E2 -27775.63} C_VEL
LIN {X 0,Y 84.181,Z 534.481,A -85,B 0,C 180,E1 -27779.939,E2 -27779.939} C_VEL
LIN {X 0,Y 80.514,Z 540.232,A -85,B 0,C 180,E1 -27786.871,E2 -27786.871} C_VEL
LIN {X 0,Y 78.162,Z 544.75,A -85,B 0,C 180,E1 -27794.35,E2 -27794.35} C_VEL
LIN {X 0,Y 77.202,Z 547.07,A -85,B 0,C 180,E1 -27799.509,E2 -27799.509} C_VEL
LIN {X 0,Y 76.675,Z 550.541,A -85,B 0,C 180,E1 -27809.999,E2 -27809.999} C_VEL
LIN {X 0,Y 77.219,Z 552.162,A -85,B 0,C 180,E1 -27820.487,E2 -27820.487} C_VEL
LIN {X 0,Y 78.235,Z 552.452,A -85,B 0,C 180,E1 -27825.634,E2 -27825.634} C_VEL
LIN {X 0,Y 81.871,Z 551.85,A -85,B 0,C 180,E1 -27835.417,E2 -27835.417} C_VEL
LIN {X 0,Y 87.744,Z 549.613,A -85,B 0,C 180,E1 -27844.102,E2 -27844.102} C_VEL
LIN {X 0,Y 93.397,Z 546.948,A -85,B 0,C 180,E1 -27849.762,E2 -27849.762} C_VEL
LIN {X 0,Y 99.722,Z 543.317,A -85,B 0,C 180,E1 -27854.81,E2 -27854.81} C_VEL
LIN {X 0,Y 106.705,Z 538.62,A -85,B 0,C 180,E1 -27859.238,E2 -27859.238} C_VEL
LIN {X 0,Y 114.411,Z 532.688,A -85,B 0,C 180,E1 -27862.992,E2 -27862.992} C_VEL
LIN {X 0,Y 121.146,Z 526.749,A -85,B 0,C 180,E1 -27865.759,E2 -27865.759} C_VEL
LIN {X 0,Y 128.156,Z 519.626,A -85,B 0,C 180,E1 -27868.213,E2 -27868.213} C_VEL
LIN {X 0,Y 135.436,Z 510.995,A -85,B 0,C 180,E1 -27870.364,E2 -27870.364} C_VEL
LIN {X 0,Y 142.132,Z 501.585,A -85,B 0,C 180,E1 -27872.112,E2 -27872.112} C_VEL
LIN {X 0,Y 147.42,Z 492.829,A -85,B 0,C 180,E1 -27873.364,E2 -27873.364} C_VEL
LIN {X 0,Y 152.769,Z 482.046,A -85,B 0,C 180,E1 -27874.533,E2 -27874.533} C_VEL
LIN {X 0,Y 156.44,Z 473.14,A -85,B 0,C 180,E1 -27875.237,E2 -27875.237} C_VEL
LIN {X 0,Y 160.239,Z 461.103,A -85,B 0,C 180,E1 -27875.914,E2 -27875.914} C_VEL
LIN {X 0,Y 162.66,Z 450.323,A -85,B 0,C 180,E1 -27876.374,E2 -27876.374} C_VEL
LIN {X 0,Y 163.607,Z 444.318,A -85,B 0,C 180,E1 -27876.607,E2 -27876.607} C_VEL
LIN {X 0,Y 163.148,Z 442.37,A -85,B 0,C 180,E1 -27877.902,E2 -27877.902} C_VEL
LIN {X 0,Y 162.282,Z 440.013,A -85,B 0,C 180,E1 -27880.225,E2 -27880.225} C_VEL
LIN {X 0,Y 161.519,Z 437.593,A -85,B 0,C 180,E1 -27883.188,E2 -27883.188} C_VEL
LIN {X 0,Y 160.984,Z 436.635,A -85,B 0,C 180,E1 -27887.392,E2 -27887.392} C_VEL
LIN {X 0,Y 161.088,Z 436.601,A -85,B 0,C 180,E1 -27890.066,E2 -27890.066} C_VEL
LIN {X 0,Y 161.154,Z 437.656,A -85,B 0,C 180,E1 -27891.41,E2 -27891.41} C_VEL
LIN {X 0,Y 161.158,Z 439.612,A -85,B 0,C 180,E1 -27892.642,E2 -27892.642} C_VEL
LIN {X 0,Y 161.142,Z 446.084,A -85,B 0,C 180,E1 -27895.75,E2 -27895.75} C_VEL
LIN {X 0,Y 161.295,Z 447.361,A -85,B 0,C 180,E1 -27896.603,E2 -27896.603} C_VEL
LIN {X 0,Y 161.479,Z 448.163,A -85,B 0,C 180,E1 -27897.27,E2 -27897.27} C_VEL
LIN {X 0,Y 159.41,Z 457.811,A -85,B 0,C 180,E1 -27897.675,E2 -27897.675} C_VEL
LIN {X 0,Y 156.916,Z 466.452,A -85,B 0,C 180,E1 -27898.092,E2 -27898.092} C_VEL
LIN {X 0,Y 153.333,Z 476.249,A -85,B 0,C 180,E1 -27898.767,E2 -27898.767} C_VEL
LIN {X 0,Y 148.468,Z 486.749,A -85,B 0,C 180,E1 -27899.724,E2 -27899.724} C_VEL
LIN {X 0,Y 143.21,Z 496.054,A -85,B 0,C 180,E1 -27900.838,E2 -27900.838} C_VEL
LIN {X 0,Y 137.146,Z 505.039,A -85,B 0,C 180,E1 -27902.228,E2 -27902.228} C_VEL
LIN {X 0,Y 130.337,Z 513.602,A -85,B 0,C 180,E1 -27904.015,E2 -27904.015} C_VEL
LIN {X 0,Y 123.982,Z 520.517,A -85,B 0,C 180,E1 -27905.902,E2 -27905.902} C_VEL
LIN {X 0,Y 115.55,Z 528.242,A -85,B 0,C 180,E1 -27908.753,E2 -27908.753} C_VEL
LIN {X 0,Y 107.76,Z 534.343,A -85,B 0,C 180,E1 -27911.963,E2 -27911.963} C_VEL
LIN {X 0,Y 101.803,Z 538.467,A -85,B 0,C 180,E1 -27914.874,E2 -27914.874} C_VEL
LIN {X 0,Y 93.439,Z 543.276,A -85,B 0,C 180,E1 -27919.918,E2 -27919.918} C_VEL
LIN {X 0,Y 85.982,Z 546.806,A -85,B 0,C 180,E1 -27925.959,E2 -27925.959} C_VEL
LIN {X 0,Y 80.891,Z 548.805,A -85,B 0,C 180,E1 -27931.42,E2 -27931.42} C_VEL
LIN {X 0,Y 74.471,Z 550.357,A -85,B 0,C 180,E1 -27941.348,E2 -27941.348} C_VEL
LIN {X 0,Y 72.099,Z 550.625,A -85,B 0,C 180,E1 -27946.974,E2 -27946.974} C_VEL
LIN {X 0,Y 70.316,Z 550.257,A -85,B 0,C 180,E1 -27953.153,E2 -27953.153} C_VEL
LIN {X 0,Y 68.878,Z 548.322,A -85,B 0,C 180,E1 -27965.913,E2 -27965.913} C_VEL
LIN {X 0,Y 69.654,Z 545.549,A -85,B 0,C 180,E1 -27975.39,E2 -27975.39} C_VEL
LIN {X 0,Y 71.793,Z 541.644,A -85,B 0,C 180,E1 -27984.383,E2 -27984.383} C_VEL
LIN {X 0,Y 75.003,Z 536.541,A -85,B 0,C 180,E1 -27992.686,E2 -27992.686} C_VEL
LIN {X 0,Y 78.445,Z 531.605,A -85,B 0,C 180,E1 -27998.686,E2 -27998.686} C_VEL
LIN {X 0,Y 83.067,Z 524.916,A -85,B 0,C 180,E1 -28004.704,E2 -28004.704} C_VEL
LIN {X 0,Y 88.298,Z 517,A -85,B 0,C 180,E1 -28009.894,E2 -28009.894} C_VEL
LIN {X 0,Y 93.247,Z 508.804,A -85,B 0,C 180,E1 -28013.899,E2 -28013.899} C_VEL
LIN {X 0,Y 98.171,Z 499.82,A -85,B 0,C 180,E1 -28017.154,E2 -28017.154} C_VEL
LIN {X 0,Y 102.656,Z 490.349,A -85,B 0,C 180,E1 -28019.759,E2 -28019.759} C_VEL
LIN {X 0,Y 106.63,Z 480.447,A -85,B 0,C 180,E1 -28021.823,E2 -28021.823} C_VEL
LIN {X 0,Y 109.905,Z 470.486,A -85,B 0,C 180,E1 -28023.403,E2 -28023.403} C_VEL
LIN {X 0,Y 112.703,Z 459.472,A -85,B 0,C 180,E1 -28024.697,E2 -28024.697} C_VEL
LIN {X 0,Y 114.843,Z 448.314,A -85,B 0,C 180,E1 -28025.541,E2 -28025.541} C_VEL
LIN {X 0,Y 117.091,Z 428.991,A -85,B 0,C 180,E1 -28026.445,E2 -28026.445} C_VEL
LIN {X 0,Y 118.134,Z 418.499,A -85,B 0,C 180,E1 -28026.898,E2 -28026.898} C_VEL
LIN {X 0,Y 117.266,Z 415.918,A -85,B 0,C 180,E1 -28027.729,E2 -28027.729} C_VEL
LIN {X 0,Y 112.501,Z 405.721,A -85,B 0,C 180,E1 -28032.286,E2 -28032.286} C_VEL
LIN {X 0,Y 108.867,Z 398.762,A -85,B 0,C 180,E1 -28036.351,E2 -28036.351} C_VEL
LIN {X 0,Y 104.808,Z 391.902,A -85,B 0,C 180,E1 -28041.74,E2 -28041.74} C_VEL
LIN {X 0,Y 102.093,Z 387.617,A -85,B 0,C 180,E1 -28046.306,E2 -28046.306} C_VEL
LIN {X 0,Y 99.785,Z 384.166,A -85,B 0,C 180,E1 -28051.201,E2 -28051.201} C_VEL
LIN {X 0,Y 99.354,Z 383.403,A -85,B 0,C 180,E1 -28052.352,E2 -28052.352} C_VEL
LIN {X 0,Y 97.215,Z 380.738,A -85,B 0,C 180,E1 -28059.881,E2 -28059.881} C_VEL
LIN {X 0,Y 96.739,Z 379.064,A -85,B 0,C 180,E1 -28064.184,E2 -28064.184} C_VEL
LIN {X 0,Y 96.627,Z 378.678,A -85,B 0,C 180,E1 -28067.396,E2 -28067.396} C_VEL
LIN {X 0,Y 97.046,Z 378.893,A -85,B 0,C 180,E1 -28073.804,E2 -28073.804} C_VEL
LIN {X 0,Y 97.431,Z 379.525,A -85,B 0,C 180,E1 -28076.165,E2 -28076.165} C_VEL
LIN {X 0,Y 98.83,Z 382.437,A -85,B 0,C 180,E1 -28081.909,E2 -28081.909} C_VEL
LIN {X 0,Y 99.89,Z 383.595,A -85,B 0,C 180,E1 -28084.673,E2 -28084.673} C_VEL
LIN {X 0,Y 102.082,Z 387.316,A -85,B 0,C 180,E1 -28089.441,E2 -28089.441} C_VEL
LIN {X 0,Y 105.131,Z 392.396,A -85,B 0,C 180,E1 -28094.555,E2 -28094.555} C_VEL
LIN {X 0,Y 108.87,Z 398.721,A -85,B 0,C 180,E1 -28099.472,E2 -28099.472} C_VEL
LIN {X 0,Y 113.383,Z 407.699,A -85,B 0,C 180,E1 -28104.453,E2 -28104.453} C_VEL
LIN {X 0,Y 115.503,Z 412.616,A -85,B 0,C 180,E1 -28106.54,E2 -28106.54} C_VEL
LIN {X 0,Y 117.947,Z 420.538,A -85,B 0,C 180,E1 -28109.024,E2 -28109.024} C_VEL
LIN {X 0,Y 114.99,Z 448.681,A -85,B 0,C 180,E1 -28110.352,E2 -28110.352} C_VEL
LIN {X 0,Y 113.327,Z 458.464,A -85,B 0,C 180,E1 -28111.064,E2 -28111.064} C_VEL
LIN {X 0,Y 110.916,Z 468.502,A -85,B 0,C 180,E1 -28112.06,E2 -28112.06} C_VEL
LIN {X 0,Y 108.103,Z 477.419,A -85,B 0,C 180,E1 -28113.171,E2 -28113.171} C_VEL
LIN {X 0,Y 104.212,Z 488.072,A -85,B 0,C 180,E1 -28115.144,E2 -28115.144} C_VEL
LIN {X 0,Y 99.694,Z 498.013,A -85,B 0,C 180,E1 -28117.525,E2 -28117.525} C_VEL
LIN {X 0,Y 95.418,Z 506.326,A -85,B 0,C 180,E1 -28120.166,E2 -28120.166} C_VEL
LIN {X 0,Y 90.309,Z 515.208,A -85,B 0,C 180,E1 -28123.957,E2 -28123.957} C_VEL
LIN {X 0,Y 86.02,Z 521.842,A -85,B 0,C 180,E1 -28127.559,E2 -28127.559} C_VEL
LIN {X 0,Y 81.351,Z 528.932,A -85,B 0,C 180,E1 -28132.789,E2 -28132.789} C_VEL
LIN {X 0,Y 76.587,Z 535.756,A -85,B 0,C 180,E1 -28139.687,E2 -28139.687} C_VEL
LIN {X 0,Y 74.009,Z 539.611,A -85,B 0,C 180,E1 -28144.701,E2 -28144.701} C_VEL
LIN {X 0,Y 71.312,Z 544.257,A -85,B 0,C 180,E1 -28152.802,E2 -28152.802} C_VEL
LIN {X 0,Y 69.843,Z 547.761,A -85,B 0,C 180,E1 -28161.318,E2 -28161.318} C_VEL
LIN {X 0,Y 69.578,Z 550.228,A -85,B 0,C 180,E1 -28169.999,E2 -28169.999} C_VEL
LIN {X 0,Y 70.233,Z 552.011,A -85,B 0,C 180,E1 -28181.544,E2 -28181.544} C_VEL
LIN {X 0,Y 73.164,Z 552.214,A -85,B 0,C 180,E1 -28192.596,E2 -28192.596} C_VEL
LIN {X 0,Y 75.491,Z 551.863,A -85,B 0,C 180,E1 -28197.741,E2 -28197.741} C_VEL
LIN {X 0,Y 81.961,Z 549.78,A -85,B 0,C 180,E1 -28206.886,E2 -28206.886} C_VEL
LIN {X 0,Y 88.037,Z 547.23,A -85,B 0,C 180,E1 -28212.731,E2 -28212.731} C_VEL
LIN {X 0,Y 94.823,Z 543.722,A -85,B 0,C 180,E1 -28217.831,E2 -28217.831} C_VEL
LIN {X 0,Y 102.234,Z 539.172,A -85,B 0,C 180,E1 -28222.237,E2 -28222.237} C_VEL
LIN {X 0,Y 111.661,Z 532.27,A -85,B 0,C 180,E1 -28226.507,E2 -28226.507} C_VEL
LIN {X 0,Y 118.78,Z 526.252,A -85,B 0,C 180,E1 -28229.085,E2 -28229.085} C_VEL
LIN {X 0,Y 126.04,Z 519.064,A -85,B 0,C 180,E1 -28231.428,E2 -28231.428} C_VEL
LIN {X 0,Y 133.64,Z 510.318,A -85,B 0,C 180,E1 -28233.381,E2 -28233.381} C_VEL
LIN {X 0,Y 139.773,Z 501.992,A -85,B 0,C 180,E1 -28234.832,E2 -28234.832} C_VEL
LIN {X 0,Y 145.991,Z 491.915,A -85,B 0,C 180,E1 -28236.157,E2 -28236.157} C_VEL
LIN {X 0,Y 150.7,Z 482.776,A -85,B 0,C 180,E1 -28237.08,E2 -28237.08} C_VEL
LIN {X 0,Y 155.214,Z 471.945,A -85,B 0,C 180,E1 -28237.852,E2 -28237.852} C_VEL
LIN {X 0,Y 158.855,Z 460.492,A -85,B 0,C 180,E1 -28238.436,E2 -28238.436} C_VEL
LIN {X 0,Y 161.159,Z 450.553,A -85,B 0,C 180,E1 -28238.827,E2 -28238.827} C_VEL
LIN {X 0,Y 161.445,Z 448.612,A -85,B 0,C 180,E1 -28238.959,E2 -28238.959} C_VEL
LIN {X 0,Y 160.804,Z 446.505,A -85,B 0,C 180,E1 -28241.197,E2 -28241.197} C_VEL
LIN {X 0,Y 160.321,Z 444.436,A -85,B 0,C 180,E1 -28243.944,E2 -28243.944} C_VEL
LIN {X 0,Y 159.973,Z 443.707,A -85,B 0,C 180,E1 -28247.311,E2 -28247.311} C_VEL
LIN {X 0,Y 160.085,Z 443.724,A -85,B 0,C 180,E1 -28250.286,E2 -28250.286} C_VEL
LIN {X 0,Y 160.539,Z 444.655,A -85,B 0,C 180,E1 -28253.402,E2 -28253.402} C_VEL
LIN {X 0,Y 161.295,Z 447.361,A -85,B 0,C 180,E1 -28256.603,E2 -28256.603} C_VEL
LIN {X 0,Y 161.253,Z 448.918,A -85,B 0,C 180,E1 -28257.063,E2 -28257.063} C_VEL
LIN {X 0,Y 160.789,Z 451.709,A -85,B 0,C 180,E1 -28257.193,E2 -28257.193} C_VEL
LIN {X 0,Y 160.16,Z 453.951,A -85,B 0,C 180,E1 -28257.047,E2 -28257.047} C_VEL
LIN {X 0,Y 156.699,Z 463.918,A -85,B 0,C 180,E1 -28255.606,E2 -28255.606} C_VEL
LIN {X 0,Y 155.317,Z 467.61,A -85,B 0,C 180,E1 -28255.586,E2 -28255.586} C_VEL
LIN {X 0,Y 151.881,Z 476.668,A -85,B 0,C 180,E1 -28256.165,E2 -28256.165} C_VEL
LIN {X 0,Y 147.069,Z 486.807,A -85,B 0,C 180,E1 -28257.009,E2 -28257.009} C_VEL
LIN {X 0,Y 141.344,Z 496.616,A -85,B 0,C 180,E1 -28258.084,E2 -28258.084} C_VEL
LIN {X 0,Y 135.298,Z 505.292,A -85,B 0,C 180,E1 -28259.336,E2 -28259.336} C_VEL
LIN {X 0,Y 128.182,Z 513.907,A -85,B 0,C 180,E1 -28261.009,E2 -28261.009} C_VEL
LIN {X 0,Y 121.378,Z 520.967,A -85,B 0,C 180,E1 -28262.81,E2 -28262.81} C_VEL
LIN {X 0,Y 112.945,Z 528.363,A -85,B 0,C 180,E1 -28265.38,E2 -28265.38} C_VEL
LIN {X 0,Y 104.786,Z 534.457,A -85,B 0,C 180,E1 -28268.399,E2 -28268.399} C_VEL
LIN {X 0,Y 97.376,Z 539.192,A -85,B 0,C 180,E1 -28271.716,E2 -28271.716} C_VEL
LIN {X 0,Y 91.025,Z 542.724,A -85,B 0,C 180,E1 -28275.18,E2 -28275.18} C_VEL
LIN {X 0,Y 82.772,Z 546.463,A -85,B 0,C 180,E1 -28280.936,E2 -28280.936} C_VEL
LIN {X 0,Y 75.76,Z 548.926,A -85,B 0,C 180,E1 -28287.636,E2 -28287.636} C_VEL
LIN {X 0,Y 68.545,Z 550.462,A -85,B 0,C 180,E1 -28297.967,E2 -28297.967} C_VEL
LIN {X 0,Y 66.475,Z 550.687,A -85,B 0,C 180,E1 -28302.264,E2 -28302.264} C_VEL
LIN {X 0,Y 63.711,Z 550.368,A -85,B 0,C 180,E1 -28310.552,E2 -28310.552} C_VEL
LIN {X 0,Y 61.827,Z 548.783,A -85,B 0,C 180,E1 -28322.956,E2 -28322.956} C_VEL
LIN {X 0,Y 62.252,Z 546.217,A -85,B 0,C 180,E1 -28333.607,E2 -28333.607} C_VEL
LIN {X 0,Y 64.327,Z 542.532,A -85,B 0,C 180,E1 -28343.728,E2 -28343.728} C_VEL
LIN {X 0,Y 68.234,Z 536.67,A -85,B 0,C 180,E1 -28354.431,E2 -28354.431} C_VEL
LIN {X 0,Y 72.194,Z 531.423,A -85,B 0,C 180,E1 -28361.228,E2 -28361.228} C_VEL
LIN {X 0,Y 76.952,Z 525.062,A -85,B 0,C 180,E1 -28367.267,E2 -28367.267} C_VEL
LIN {X 0,Y 82.427,Z 517.337,A -85,B 0,C 180,E1 -28372.563,E2 -28372.563} C_VEL
LIN {X 0,Y 87.862,Z 508.849,A -85,B 0,C 180,E1 -28376.821,E2 -28376.821} C_VEL
LIN {X 0,Y 92.988,Z 500.016,A -85,B 0,C 180,E1 -28380.048,E2 -28380.048} C_VEL
LIN {X 0,Y 97.701,Z 490.569,A -85,B 0,C 180,E1 -28382.65,E2 -28382.65} C_VEL
LIN {X 0,Y 101.525,Z 481.565,A -85,B 0,C 180,E1 -28384.562,E2 -28384.562} C_VEL
LIN {X 0,Y 105.415,Z 470.307,A -85,B 0,C 180,E1 -28386.32,E2 -28386.32} C_VEL
LIN {X 0,Y 108.327,Z 459.235,A -85,B 0,C 180,E1 -28387.588,E2 -28387.588} C_VEL
LIN {X 0,Y 110.412,Z 448.884,A -85,B 0,C 180,E1 -28388.354,E2 -28388.354} C_VEL
LIN {X 0,Y 112.721,Z 430.063,A -85,B 0,C 180,E1 -28389.217,E2 -28389.217} C_VEL
LIN {X 0,Y 113.61,Z 420.549,A -85,B 0,C 180,E1 -28389.689,E2 -28389.689} C_VEL
LIN {X 0,Y 109.367,Z 410.904,A -85,B 0,C 180,E1 -28394.199,E2 -28394.199} C_VEL
LIN {X 0,Y 106.197,Z 404.459,A -85,B 0,C 180,E1 -28398.132,E2 -28398.132} C_VEL
LIN {X 0,Y 102.793,Z 398.244,A -85,B 0,C 180,E1 -28403.12,E2 -28403.12} C_VEL
LIN {X 0,Y 100.076,Z 393.798,A -85,B 0,C 180,E1 -28408.15,E2 -28408.15} C_VEL
LIN {X 0,Y 98.06,Z 390.263,A -85,B 0,C 180,E1 -28413.169,E2 -28413.169} C_VEL
LIN {X 0,Y 96.06,Z 387.417,A -85,B 0,C 180,E1 -28421.134,E2 -28421.134} C_VEL
LIN {X 0,Y 95.739,Z 385.99,A -85,B 0,C 180,E1 -28425.098,E2 -28425.098} C_VEL
LIN {X 0,Y 95.848,Z 385.686,A -85,B 0,C 180,E1 -28431.566,E2 -28431.566} C_VEL
LIN {X 0,Y 96.293,Z 386.315,A -85,B 0,C 180,E1 -28435.121,E2 -28435.121} C_VEL
LIN {X 0,Y 97.419,Z 389.045,A -85,B 0,C 180,E1 -28440.534,E2 -28440.534} C_VEL
LIN {X 0,Y 98.442,Z 390.374,A -85,B 0,C 180,E1 -28443.58,E2 -28443.58} C_VEL
LIN {X 0,Y 100.823,Z 394.77,A -85,B 0,C 180,E1 -28449.117,E2 -28449.117} C_VEL
LIN {X 0,Y 103.182,Z 399.01,A -85,B 0,C 180,E1 -28453.352,E2 -28453.352} C_VEL
LIN {X 0,Y 105.805,Z 403.699,A -85,B 0,C 180,E1 -28457.164,E2 -28457.164} C_VEL
LIN {X 0,Y 109.205,Z 410.696,A -85,B 0,C 180,E1 -28461.454,E2 -28461.454} C_VEL
LIN {X 0,Y 111.759,Z 416.731,A -85,B 0,C 180,E1 -28464.319,E2 -28464.319} C_VEL
LIN {X 0,Y 113.503,Z 422.632,A -85,B 0,C 180,E1 -28466.296,E2 -28466.296} C_VEL
LIN {X 0,Y 110.723,Z 447.917,A -85,B 0,C 180,E1 -28467.458,E2 -28467.458} C_VEL
LIN {X 0,Y 109.009,Z 457.865,A -85,B 0,C 180,E1 -28468.152,E2 -28468.152} C_VEL
LIN {X 0,Y 106.691,Z 467.421,A -85,B 0,C 180,E1 -28469.055,E2 -28469.055} C_VEL
LIN {X 0,Y 103.661,Z 476.853,A -85,B 0,C 180,E1 -28470.182,E2 -28470.182} C_VEL
LIN {X 0,Y 99.579,Z 487.592,A -85,B 0,C 180,E1 -28472.12,E2 -28472.12} C_VEL
LIN {X 0,Y 94.848,Z 497.598,A -85,B 0,C 180,E1 -28474.478,E2 -28474.478} C_VEL
LIN {X 0,Y 89.732,Z 506.998,A -85,B 0,C 180,E1 -28477.531,E2 -28477.531} C_VEL
LIN {X 0,Y 85.474,Z 514.016,A -85,B 0,C 180,E1 -28480.485,E2 -28480.485} C_VEL
LIN {X 0,Y 79.786,Z 522.33,A -85,B 0,C 180,E1 -28485.195,E2 -28485.195} C_VEL
LIN {X 0,Y 74.822,Z 529.265,A -85,B 0,C 180,E1 -28490.652,E2 -28490.652} C_VEL
LIN {X 0,Y 70.532,Z 535.042,A -85,B 0,C 180,E1 -28496.767,E2 -28496.767} C_VEL
LIN {X 0,Y 66.458,Z 540.616,A -85,B 0,C 180,E1 -28504.975,E2 -28504.975} C_VEL
LIN {X 0,Y 63.827,Z 544.983,A -85,B 0,C 180,E1 -28514.021,E2 -28514.021} C_VEL
